END_IF
END_FUNCTION_BLOCK
ACTION CachePointers:
;
END_ACTION
ACTION CheckUpdateFlags:
xDataInUpdated := TRUE;
END_ACTION
ACTION DataReceived:
cmd := InDataTelegram_Module_1[0];
IF (cmd = M2C_NVI_UPDT_OCCD) OR (cmd = M2C_NV_VALUE_RSP) OR (cmd = M2C_NVI_UPDT_TOUT) THEN
	bNvRelativeIdx := (InDataTelegram_Module_1[1] - bNvStartIndex - bObjectIndex) / bLmoCount;
	CASE bNvRelativeIdx OF

	END_CASE
ELSIF (cmd = M2C_CP_VALUE_RSP) THEN
	wCpRelativeIdx := ((InDataTelegram_Module_1[1] + InDataTelegram_Module_1[2] * 256) - wCpStartIndex - bObjectIndex) / bLmoCount;
	CASE wCpRelativeIdx OF

	END_CASE
END_IF
END_ACTION
ACTION ResetNviUpdate:
;
END_ACTION
ACTION SendValueRequest:
;
END_ACTION
ACTION SetUpdateFlags:
;
END_ACTION

(* POU Plant/SCA_Proc, ST *)
PROGRAM SCA_Proc
VAR
	SCA01_1	:	FLT_TAP;
	SCA01_2	:	FLT_TAP;
	SCA01_3	:	FLT_TAP;

	upd		:	BOOL;
END_VAR
(***** SCA01 *****)
SCA01_1(IN:=SCA01_1_DI);
IF SCA01_1.EVL THEN LogEv(EL_Wrn,EO_SCA,1,1,'1'); upd:=TRUE; END_IF
IF SCA01_1.EVH THEN	LogEv(EL_Log,EO_SCA,1,2,'1'); upd:=TRUE; END_IF

SCA01_2(IN:=SCA01_2_DI);
IF SCA01_2.EVL THEN	LogEv(EL_Wrn,EO_SCA,1,1,'2'); upd:=TRUE; END_IF
IF SCA01_2.EVH THEN	LogEv(EL_Log,EO_SCA,1,2,'2'); upd:=TRUE; END_IF

SCA01_3(IN:=SCA01_3_DI);
IF SCA01_3.EVL THEN	LogEv(EL_Wrn,EO_SCA,1,1,'3'); upd:=TRUE; END_IF
IF SCA01_3.EVH THEN	LogEv(EL_Log,EO_SCA,1,2,'3'); upd:=TRUE; END_IF

IF upd THEN
	upd:=FALSE;
	Logger_Head();
	AddLogData();
	Logger_Send();
END_IF
END_PROGRAM
ACTION AddLogData:
Logger.s1:='&SCA01=';
Logger.s1:=CONCAT(Logger.s1,BYTE_TO_STRING(BOOL_TO_BYTE(SCA01_1.OUT))		); Logger.s1:=CONCAT(Logger.s1,';');
Logger.s1:=CONCAT(Logger.s1,BYTE_TO_STRING(BOOL_TO_BYTE(SCA01_2.OUT))		); Logger.s1:=CONCAT(Logger.s1,';');
Logger.s1:=CONCAT(Logger.s1,BYTE_TO_STRING(BOOL_TO_BYTE(SCA01_3.OUT))		);
ADDSTRING(ADR(Logger.TData), ADR(Logger.s1), Logger.TLen);
END_ACTION

(* POU TCP_Logger/LogEv, ST *)
FUNCTION LogEv : BOOL
VAR_INPUT
	Level	: en_Logger_ErrLev;
	Object  : en_SYS_Objects;
	Index	: WORD;
	Error	: WORD;
	Message : STRING;
END_VAR
VAR
	s1 : STRING(160);
	i  : INT;
END_VAR
(* Execute error level operations *)
CASE Level OF
	EL_Wrn: 		Sys.Warning:=TRUE;
	EL_Alarm: 		Sys.Alarm  :=TRUE;
	EL_AlarmStop: 	Sys.Alarm  :=TRUE; (* GO TO STOP STATE!! *)
END_CASE

(* Fill lastlog list *)
s1:=CONCAT(Sys.Time_LogString,';Lev=');
s1:=CONCAT(s1,INT_TO_STRING(Level));
s1:=CONCAT(s1,';Obj=');
s1:=CONCAT(s1,INT_TO_STRING(Object));
s1:=CONCAT(s1,';Idx=');
s1:=CONCAT(s1,WORD_TO_STRING(Index));
s1:=CONCAT(s1,';Err=');
s1:=CONCAT(s1,WORD_TO_STRING(Error));
Sys.LastLogs_Dat[Sys.LastLogs_Idx]:=s1;
Sys.LastLogs_Msg[Sys.LastLogs_Idx]:=Message;
Sys.LastLogs_Idx:=Sys.LastLogs_Idx+1;
IF Sys.LastLogs_Idx>5 THEN Sys.LastLogs_Idx:=0; END_IF

(*---------------------------------------------------------------*)
	Logger_Head();
(*---------------------------------------------------------------*)

(* Insert ERR *)
s1:=CONCAT('&ERR=',INT_TO_STRING(Level));
s1:=CONCAT(s1,';');
s1:=CONCAT(s1,INT_TO_STRING(Object));
s1:=CONCAT(s1,';');
s1:=CONCAT(s1,WORD_TO_STRING(Index));
s1:=CONCAT(s1,';');
s1:=CONCAT(s1,WORD_TO_STRING(Error));
s1:=CONCAT(s1,';');
ADDSTRING(ADR(Logger.TData), ADR(s1), Logger.TLen);
s1:=Message;
STR_NOSPACES(ADR(s1));
ADDSTRING(ADR(Logger.TData), ADR(s1), Logger.TLen);

(*---------------------------------------------------------------*)
	Logger_Send();
(*---------------------------------------------------------------*)
END_FUNCTION

(* POU TCP_Logger/Logger_Head, ST *)
FUNCTION Logger_Head : BOOL
VAR
	s1 : STRING(160);
	i  : BYTE;
END_VAR
Logger.TLen:=0;
(* Set GET header *)
ADDSTRING(ADR(Logger.TData), ADR(Logger_GETSTART), Logger.TLen);

(* Insert Header *)
s1:=INSERT('ID=&V=1&D=',DWORD_TO_STRING(Plant_SN),3);
s1:=CONCAT(s1,Sys.Time_LogString);
s1:=CONCAT(s1,'&S=');
IF Sys.Alarm THEN i:=2; ELSIF Sys.Warning THEN i:=1; ELSE i:=0; END_IF
s1:=CONCAT(s1,BYTE_TO_STRING(i));
ADDSTRING(ADR(Logger.TData), ADR(s1), Logger.TLen);
END_FUNCTION

(* POU Utils Functions/ADDSTRING, ST *)
FUNCTION ADDSTRING : BOOL (* Append string to a byte buffer *)
VAR_INPUT
	pTxData: POINTER TO BYTE;
	pString: POINTER TO BYTE;
END_VAR
VAR_IN_OUT
	TxLen: DINT;
END_VAR
VAR
END_VAR
pTxData:=pTxData+TxLen;
WHILE pString^<>0 DO
	pTxData^:=pString^;
	pString:=pString+1;
	pTxData:=pTxData+1;
	TxLen:=TxLen+1;
END_WHILE
END_FUNCTION

(* POU Utils Functions/STR_NOSPACES, ST *)
FUNCTION STR_NOSPACES : BOOL (* Replace spaces and bad chars with allowed ones, used as HTTP-GET validator *)
VAR_INPUT
	pString: POINTER TO BYTE;
END_VAR
VAR
END_VAR
WHILE pString^<>0 DO
	IF pString^=16#20 (* space *) THEN pString^:=16#5F; (*'_'*) END_IF
	pString:=pString+1;
END_WHILE
END_FUNCTION

(* POU TCP_Logger/Logger_Send, ST *)
FUNCTION Logger_Send : BOOL
VAR
	hFile: 	DWORD;
	pos:	DWORD;
END_VAR
(* Finalize string *)
ADDSTRING(ADR(Logger.TData), ADR(Logger_GETEND), Logger.TLen);

(* Read log position *)
pos:=SysFileGetSize(Logger_DataFile);
(* Check log size, bckup and erase if no pending messages *)
IF pos>5000000(*5M*) THEN
	hFile:=SysFileOpen(Logger_IndexFile,'r');
	IF hFile=0 THEN
		SysFileDelete(Logger_DataFileOld);
		SysFileRename(Logger_DataFile,Logger_DataFileOld);
		pos:=0;
	ELSE
		SysFileClose(hFile);
	END_IF
END_IF
(* Write message on log file *)
hFile:=SysFileOpen(Logger_DataFile,'a');
IF hFile<>0 THEN
	SysFileWrite(hFile, ADR(Logger.TData), Logger.TLen);
	SysFileClose(hFile);
ELSE
	Sys.Warning:=TRUE;
END_IF


(* Check logger status *)
IF Logger.SendReq=FALSE THEN
	(* Set log position for recovery *)
	Logger.SendIdx:=pos;
	(* Copy message data *)
	MEMCPY(ADR(Logger.TData),ADR(Logger.SendData),DINT_TO_WORD(Logger.TLen));
	Logger.SendLen:=Logger.TLen;
	(* Trigger request *)
	Logger.SendReq:=TRUE;
ELSE
	(* Add message position+size in recovery indexes *)
	hFile:=SysFileOpen(Logger_IndexFile,'a');
	SysFileWrite(hFile, ADR(pos), SIZEOF(pos));
	SysFileWrite(hFile, ADR(Logger.TLen), SIZEOF(Logger.TLen));
	SysFileClose(hFile);
END_IF
END_FUNCTION

(* POU Utils Functions/MEMCPY, ST *)
FUNCTION MEMCPY:BOOL
VAR_INPUT
	pSourceAddress:POINTER TO ARRAY[1..2] OF BYTE;
	pDestinationAddress:POINTER TO ARRAY[1..2] OF BYTE;
	BytesToCopy:WORD;
END_VAR
VAR
END_VAR
WHILE (BytesToCopy > 0) DO
	pDestinationAddress^[1]:=pSourceAddress^[1]; (* copy bytes from source to destination *)
	pDestinationAddress:=ADR(pDestinationAddress^[2]); (* increment destination *)
	pSourceAddress:=ADR(pSourceAddress^[2]);(* increment source *)
	BytesToCopy:=BytesToCopy -1; (* decrement number of bytes to copy *)
END_WHILE
END_FUNCTION

(* POU Plant/SYS_Proc, ST *)
PROGRAM SYS_Proc
VAR
(*	fALARM_PB		:FLT_TAP;
	fALARM_TB		:FLT_TAP;
	fALARM_PM		:FLT_TAP; *)

(*	fGZB_ST			:FLT_TAP; (* GATEWAY ZIGBEE *)*)
(*	fVPN_OUT1		:FLT_TAP; (* VPN - CONNECT *)*)
	fVPN_OUT2		:FLT_TAP; (* VPN - STATUS *)
(*	fKEY_CT_ST		:FLT_TAP; (* DOOR01 - Porta primaria *)*)
(*	fKEY_SCT_ST		:FLT_TAP; (* DOOR02 - Porta secondaria *)*)
	fKEY_QE_ST		:FLT_TAP; (* DOOR03 - Quadro Elettrico *)
	fKEY_ManualMode :FLT_TAP; (* Selettore Luci in manuale *)

END_VAR
(*************** ISPESL *****************)
(*
fALARM_PB(IN:=ALARM_PB);
IF fALARM_PB.EVH THEN
	LogEv(EL_AlarmStop,EO_PBV,1,1,'Over_Pressure_Alarm');
END_IF

fALARM_TB(IN:=ALARM_TB);
IF fALARM_TB.EVH THEN
	LogEv(EL_AlarmStop,EO_TBV,1,1,'Over_Temperature_Alarm');
END_IF

fALARM_PM(IN:=ALARM_PM);
IF fALARM_PM.EVH THEN
	LogEv(EL_AlarmStop,EO_PMV,1,1,'Under_Pressure_Alarm');
END_IF
*)
(****************************************)

(*### VPN Connection Check ###*)(*
fVPN_OUT1(IN:=VPN_OUT1);
IF fVPN_OUT1.EVH THEN
	LogEv(EL_Log,EO_VPN,1,1,'CONNECT_ON');
END_IF
IF fVPN_OUT1.EVL THEN
	LogEv(EL_Log,EO_VPN,1,2,'CONNECT_OFF');
END_IF*)

(*### VPN Status Check ###*)
fVPN_OUT2(IN:=VPN_OUT2);
IF fVPN_OUT2.EVH THEN
	LogEv(EL_Log,EO_VPN,1,3,'STATUS_UP');
END_IF
IF fVPN_OUT2.EVL THEN
	LogEv(EL_Wrn,EO_VPN,1,4,'STATUS_DOWN');
END_IF

(*### DOOR01 Status Check ###*)(*
fKEY_CT_ST(IN:=KEY_CT_ST);
IF fKEY_CT_ST.EVH THEN
	LogEv(EL_Log,EO_DOOR,1,2,'Centrale_termica_Close');
END_IF
IF fKEY_CT_ST.EVL THEN
	LogEv(EL_Wrn,EO_DOOR,1,1,'Centrale_termica_Open');
END_IF*)

(*### DOOR02 Status Check ###*)(*
fKEY_SCT_ST(IN:=KEY_SCT_ST);
IF fKEY_SCT_ST.EVH THEN
	LogEv(EL_Log,EO_DOOR,2,2,'Sottocentrale_termica_Close');
END_IF
IF fKEY_SCT_ST.EVL THEN
	LogEv(EL_Wrn,EO_DOOR,2,1,'Sottocentrale_termica_Open');
END_IF*)

(*### DOOR03 Status Check ###*)
fKEY_QE_ST(IN:=KEY_QE_ST);
IF fKEY_QE_ST.EVH THEN
	LogEv(EL_Log,EO_DOOR,3,2,'Quadro_Close');
END_IF
IF fKEY_QE_ST.EVL THEN
	LogEv(EL_Wrn,EO_DOOR,3,1,'Quadro_Open');
END_IF

(*### Selettore luci in manuale ###*)
fKEY_ManualMode(IN:=SCA01_1_DI);
IF fKEY_ManualMode.EVH THEN
	LogEv(EL_Alarm,EO_LUX,0,10,'Impianto_in Manuale');
END_IF
IF fKEY_ManualMode.EVL THEN
	LogEv(EL_Log,EO_LUX,0,11,'Impianto_In_Automatico');
END_IF
END_PROGRAM

(* POU Utils Functions/AVERAGE_T, ST *)
FUNCTION_BLOCK AVERAGE_T
VAR_INPUT
	IN: 	INT;
END_VAR
VAR_OUTPUT
	HI:		INT;
	AVG:	INT;
	LOW:	INT;
	ERR:	BOOL;
END_VAR
VAR
	sum:	DINT;
	cnt:	WORD;
END_VAR
IF cnt>=65000 THEN
	ERR:=TRUE;
	Read();
	sum := sum - AVG;
	cnt := cnt + 1;
END_IF

sum := sum + IN;
cnt := cnt + 1;

IF IN<LOW THEN  LOW:=IN; END_IF
IF IN>HI  THEN HI :=IN; END_IF
END_FUNCTION_BLOCK
ACTION Read:
AVG := DINT_TO_INT(sum/cnt);
END_ACTION
ACTION Reset:
HI:=IN;
AVG:=IN;
LOW:=IN;
ERR:=FALSE;

sum:=IN;
cnt:=1;
END_ACTION

(* POU Utils Functions/BUILD_16TO32, ST *)
FUNCTION BUILD_16TO32 : DWORD
VAR_INPUT
		pSource	:	POINTER TO WORD;
END_VAR
VAR
		Data	:	DWORD;
END_VAR
Data := WORD_TO_DWORD(pSource^);
pSource := pSource + 1;
Data := Data + WORD_TO_DWORD(pSource^) * 65536;

BUILD_16TO32 := Data;
END_FUNCTION

(* POU Utils Functions/COPY_32SWAP16, ST *)
FUNCTION COPY_32SWAP16:BOOL
VAR_INPUT
	pSourceAddress		:POINTER TO ARRAY[1..2] OF WORD;
	pDestinationAddress	:POINTER TO ARRAY[1..2] OF WORD;
END_VAR
VAR
END_VAR
pDestinationAddress^[1]:=pSourceAddress^[2];
pDestinationAddress^[2]:=pSourceAddress^[1];
END_FUNCTION

(* POU Utils Functions/FLT_KEY, ST *)
FUNCTION_BLOCK FLT_KEY
VAR_INPUT
	IN		: BOOL;
	TTAP	: TIME:=T#5s;
	INITEV	: BOOL:=TRUE;
END_VAR
VAR_OUTPUT
	OUT		: BOOL;
	EVH		: BOOL;
	EVL		: BOOL;
END_VAR
VAR
	init	: BOOL:=FALSE;
	timer	: TON;
	timerIn	: TON;				(* Inhibition timer *)
	fInhibit: BOOL:=FALSE;
END_VAR
EVH:=FALSE;
EVL:=FALSE;

IF NOT init THEN
	init := TRUE;
	IF INITEV THEN
		OUT  := NOT IN;
	ELSE
		OUT  := IN;
	END_IF
END_IF

timerIn(IN:=fInhibit,PT:=T#500ms);

IF timerIn.Q THEN fInhibit := FALSE; END_IF

IF NOT fInhibit THEN

	IF OUT<>IN THEN
		timer(IN:=TRUE,PT:=TTAP);
		IF timer.Q THEN
			OUT:=IN;
			timer(IN:=FALSE);
			fInhibit := TRUE;
			IF OUT THEN EVH:=TRUE; ELSE EVL:=TRUE; END_IF
		END_IF
	ELSE
		timer(IN:=FALSE);
	END_IF
END_IF
END_FUNCTION_BLOCK

(* POU Utils Functions/FLT_TIME, ST *)
FUNCTION_BLOCK FLT_TIME
VAR_INPUT
	IN		: BOOL;
	TTAP	: TIME:=T#5s;
	INITEV	: BOOL:=TRUE;
END_VAR
VAR_OUTPUT
	OUT		: BOOL;
	EVH		: BOOL;
	EVL		: BOOL;
END_VAR
VAR
	init	: BOOL:=FALSE;
	timer	: TON;
END_VAR
EVH:=FALSE;
EVL:=FALSE;

IF NOT init THEN
	init := TRUE;
	IF INITEV THEN
		OUT  := NOT IN;
	ELSE
		OUT  := IN;
	END_IF
END_IF

IF OUT<>IN THEN
	timer(IN:=TRUE,PT:=TTAP);
	IF timer.Q THEN
		OUT:=IN;
		timer(IN:=FALSE);
		IF OUT THEN EVH:=TRUE; ELSE EVL:=TRUE; END_IF
	END_IF
ELSE
	timer(IN:=FALSE);
END_IF
END_FUNCTION_BLOCK

(* POU LON/Module_1/Internal/FuDoCpUpdate_Module_1, ST *)
FUNCTION FuDoCpUpdate_Module_1 : BOOL
(******************************************)
(* Automatic generated code, do not edit! *)
(******************************************)
VAR_INPUT
	ptCp : POINTER TO BYTE;
	ptCpLast : POINTER TO BYTE;
	wCpIndex : WORD;
	uiCpLength : UINT;
	uiCpVariableLength : UINT;
END_VAR
OutDataTelegram_Module_1[0] := C2M_CP_VALUE;
OutDataTelegram_Module_1[1] := WORD_TO_BYTE(wCpIndex AND 16#FF);
OutDataTelegram_Module_1[2] := WORD_TO_BYTE((wCpIndex / 256) AND 16#FF);

mbxModule_1.bTxPrio := 1;
mbxModule_1.bTxProtID := 0;
mbxModule_1.pbTxData := ADR(OutDataTelegram_Module_1);
mbxModule_1.unTxLen := 3 + uiCpLength;
mbxModule_1.MBX_SEND();

IF (mbxModule_1.nError <> MBX_OK) THEN
	FuDoCpUpdate_Module_1 := FALSE;
	RETURN;
END_IF

FuMemCopy(ptCp, ptCpLast, uiCpVariableLength);

FuDoCpUpdate_Module_1 := TRUE;
END_FUNCTION

(* POU LON/Shared/Internal/FuRawToSnvtFilePos, ST *)
FUNCTION FuRawToSnvtFilePos : BOOL
(******************************************)
(* Automatic generated code, do not edit! *)
(******************************************)
VAR_INPUT
	RawDataIn : POINTER TO ARRAY[0..5] OF BYTE;
	DataOut : POINTER TO typSnvtFilePos;
END_VAR
VAR
END_VAR
DataOut^.diRwPtr := RawDataIn^[0] * 16777216 + RawDataIn^[1] * 65536 + RawDataIn^[2] * 256 + RawDataIn^[3];

DataOut^.wRwLength := RawDataIn^[4] * 256 + RawDataIn^[5];

FuRawToSnvtFilePos := TRUE;
END_FUNCTION

(* POU LON/Shared/Internal/FuRawToSnvtFileReq, ST *)
FUNCTION FuRawToSnvtFileReq : BOOL
(******************************************)
(* Automatic generated code, do not edit! *)
(******************************************)
VAR_INPUT
	RawDataIn : POINTER TO ARRAY[0..11] OF BYTE;
	DataOut : POINTER TO typSnvtFileReq;
END_VAR
VAR
END_VAR
DataOut^.bRequest := RawDataIn^[0];

DataOut^.wIndex := RawDataIn^[1] * 256 + RawDataIn^[2];

DataOut^.wReceiveTimeout := RawDataIn^[3] * 256 + RawDataIn^[4];

DataOut^.abDestAddress[0] := RawDataIn^[5];
DataOut^.abDestAddress[1] := RawDataIn^[6];
DataOut^.abDestAddress[2] := RawDataIn^[7];
DataOut^.abDestAddress[3] := RawDataIn^[8];
DataOut^.abDestAddress[4] := RawDataIn^[9];

DataOut^.bAuthOn := RawDataIn^[10];

DataOut^.bPrioOn := RawDataIn^[11];

FuRawToSnvtFileReq := TRUE;
END_FUNCTION

(* POU LON/Shared/Internal/FuRawToSnvtFileStatus, ST *)
FUNCTION FuRawToSnvtFileStatus : BOOL
(******************************************)
(* Automatic generated code, do not edit! *)
(******************************************)
VAR_INPUT
	RawDataIn : POINTER TO ARRAY[0..26] OF BYTE;
	DataOut : POINTER TO typSnvtFileStatus;
END_VAR
VAR
END_VAR
DataOut^.bStatus := RawDataIn^[0];

DataOut^.wNumberOfFiles := RawDataIn^[1] * 256 + RawDataIn^[2];

DataOut^.wSelectedFile := RawDataIn^[3] * 256 + RawDataIn^[4];

DataOut^.abAdr[0] := RawDataIn^[5];
DataOut^.abAdr[1] := RawDataIn^[6];
DataOut^.abAdr[2] := RawDataIn^[7];
DataOut^.abAdr[3] := RawDataIn^[8];
DataOut^.abAdr[4] := RawDataIn^[9];
DataOut^.abAdr[5] := RawDataIn^[10];
DataOut^.abAdr[6] := RawDataIn^[11];
DataOut^.abAdr[7] := RawDataIn^[12];
DataOut^.abAdr[8] := RawDataIn^[13];
DataOut^.abAdr[9] := RawDataIn^[14];
DataOut^.abAdr[10] := RawDataIn^[15];
DataOut^.abAdr[11] := RawDataIn^[16];
DataOut^.abAdr[12] := RawDataIn^[17];
DataOut^.abAdr[13] := RawDataIn^[18];
DataOut^.abAdr[14] := RawDataIn^[19];
DataOut^.abAdr[15] := RawDataIn^[20];
DataOut^.abAdr[16] := RawDataIn^[21];
DataOut^.abAdr[17] := RawDataIn^[22];
DataOut^.abAdr[18] := RawDataIn^[23];
DataOut^.abAdr[19] := RawDataIn^[24];
DataOut^.abAdr[20] := RawDataIn^[25];
DataOut^.abAdr[21] := RawDataIn^[26];

FuRawToSnvtFileStatus := TRUE;
END_FUNCTION

(* POU LON/Shared/Internal/FuRawToSnvtObjRequest, ST *)
FUNCTION FuRawToSnvtObjRequest : BOOL
(******************************************)
(* Automatic generated code, do not edit! *)
(******************************************)
VAR_INPUT
	RawDataIn : POINTER TO ARRAY[0..2] OF BYTE;
	DataOut : POINTER TO typSnvtObjRequest;
END_VAR
VAR
END_VAR
DataOut^.wObjectId := RawDataIn^[0] * 256 + RawDataIn^[1];

DataOut^.bObjectRequest := RawDataIn^[2];

FuRawToSnvtObjRequest := TRUE;
END_FUNCTION

(* POU LON/Shared/Internal/FuRawToSnvtObjStatus, ST *)
FUNCTION FuRawToSnvtObjStatus : BOOL
(******************************************)
(* Automatic generated code, do not edit! *)
(******************************************)
VAR_INPUT
	RawDataIn : POINTER TO ARRAY[0..5] OF BYTE;
	DataOut : POINTER TO typSnvtObjStatus;
END_VAR
VAR
END_VAR
DataOut^.wObjectId := RawDataIn^[0] * 256 + RawDataIn^[1];

DataOut^.bBitfieldByteOffset2 := RawDataIn^[2];

DataOut^.bBitfieldByteOffset3 := RawDataIn^[3];

DataOut^.bBitfieldByteOffset4 := RawDataIn^[4];

DataOut^.bBitfieldByteOffset5 := RawDataIn^[5];

FuRawToSnvtObjStatus := TRUE;
END_FUNCTION

(* POU LON/Module_1/Internal/FuSendCpValueReq_Module_1, ST *)
FUNCTION FuSendCpValueReq_Module_1 : BOOL
(******************************************)
(* Automatic generated code, do not edit! *)
(******************************************)
VAR_INPUT
	ptCp : POINTER TO BYTE;
	ptInternalUseOnly : POINTER TO BYTE;
	wCpIndex : WORD;
END_VAR
IF (ptCp <> 0) THEN
	IF ptInternalUseOnly^.0 = TRUE THEN
		OutDataTelegram_Module_1[0] := C2M_CP_VALUE_QRY;
		OutDataTelegram_Module_1[1] := WORD_TO_BYTE(wCpIndex AND 16#FF);
		OutDataTelegram_Module_1[2] := WORD_TO_BYTE((wCpIndex / 256) AND 16#FF);

		mbxModule_1.bTxPrio := 1;
		mbxModule_1.bTxProtID := 0;
		mbxModule_1.pbTxData := ADR(OutDataTelegram_Module_1);
		mbxModule_1.unTxLen := 3;
		mbxModule_1.MBX_SEND();

		IF (mbxModule_1.nError <> MBX_OK) THEN
			FuSendCpValueReq_Module_1 := FALSE;
			RETURN;
		END_IF
		ptInternalUseOnly^.0 := FALSE;
	END_IF
END_IF

FuSendCpValueReq_Module_1 := TRUE;
END_FUNCTION

(* POU LON/Shared/Internal/FuSnvtFilePosToRaw, ST *)
FUNCTION FuSnvtFilePosToRaw : BOOL
(******************************************)
(* Automatic generated code, do not edit! *)
(******************************************)
VAR_INPUT
	NvDataIn :  POINTER TO typSnvtFilePos;
	DataOut : POINTER TO ARRAY[0..5] OF BYTE;
END_VAR
VAR
END_VAR
DataOut^[0] := DINT_TO_BYTE(SHR(NvDataIn^.diRwPtr, 24));
DataOut^[1] := DINT_TO_BYTE(SHR(NvDataIn^.diRwPtr, 16));
DataOut^[2] := DINT_TO_BYTE(SHR(NvDataIn^.diRwPtr, 8));
DataOut^[3] := DINT_TO_BYTE(NvDataIn^.diRwPtr);

DataOut^[4] := WORD_TO_BYTE(SHR(NvDataIn^.wRwLength, 8));
DataOut^[5] := WORD_TO_BYTE(NvDataIn^.wRwLength);

FuSnvtFilePosToRaw := TRUE;
END_FUNCTION

(* POU LON/Shared/Internal/FuSnvtFileReqToRaw, ST *)
FUNCTION FuSnvtFileReqToRaw : BOOL
(******************************************)
(* Automatic generated code, do not edit! *)
(******************************************)
VAR_INPUT
	NvDataIn :  POINTER TO typSnvtFileReq;
	DataOut : POINTER TO ARRAY[0..11] OF BYTE;
END_VAR
VAR
END_VAR
DataOut^[0] := NvDataIn^.bRequest;

DataOut^[1] := WORD_TO_BYTE(SHR(NvDataIn^.wIndex, 8));
DataOut^[2] := WORD_TO_BYTE(NvDataIn^.wIndex);

DataOut^[3] := WORD_TO_BYTE(SHR(NvDataIn^.wReceiveTimeout, 8));
DataOut^[4] := WORD_TO_BYTE(NvDataIn^.wReceiveTimeout);

DataOut^[5] := NvDataIn^.abDestAddress[0];
DataOut^[6] := NvDataIn^.abDestAddress[1];
DataOut^[7] := NvDataIn^.abDestAddress[2];
DataOut^[8] := NvDataIn^.abDestAddress[3];
DataOut^[9] := NvDataIn^.abDestAddress[4];

DataOut^[10] := NvDataIn^.bAuthOn;

DataOut^[11] := NvDataIn^.bPrioOn;

FuSnvtFileReqToRaw := TRUE;
END_FUNCTION

(* POU LON/Shared/Internal/FuSnvtObjRequestToRaw, ST *)
FUNCTION FuSnvtObjRequestToRaw : BOOL
(******************************************)
(* Automatic generated code, do not edit! *)
(******************************************)
VAR_INPUT
	NvDataIn :  POINTER TO typSnvtObjRequest;
	DataOut : POINTER TO ARRAY[0..2] OF BYTE;
END_VAR
VAR
END_VAR
DataOut^[0] := WORD_TO_BYTE(SHR(NvDataIn^.wObjectId, 8));
DataOut^[1] := WORD_TO_BYTE(NvDataIn^.wObjectId);

DataOut^[2] := NvDataIn^.bObjectRequest;

FuSnvtObjRequestToRaw := TRUE;
END_FUNCTION

(* POU TCP_Logger/LogTrig, ST *)
FUNCTION LogTrig : BOOL
VAR
	s1 : STRING(160);
	i  : BYTE;
END_VAR
(*---------------------------------------------------------------*)
	Logger_Head();
(*---------------------------------------------------------------*)

(* Insert contabilizers  *)
ANZ01.AddLogData( ModBus:=MODB01 );
ANZ02.AddLogData( ModBus:=MODB01 );
HVAC01.AddLogData(ModBus:=MODB02);
HVAC02.AddLogData(ModBus:=MODB02);

COOV01.AddLogData();

LUX01.AddLogData(WORKINGTIME:=LuxWT[1], POWERONCYCLES:=LuxPOC[1]);
LUX02.AddLogData(WORKINGTIME:=LuxWT[2], POWERONCYCLES:=LuxPOC[2]);
LUX03.AddLogData(WORKINGTIME:=LuxWT[3], POWERONCYCLES:=LuxPOC[3]);
LUX04.AddLogData(WORKINGTIME:=LuxWT[4], POWERONCYCLES:=LuxPOC[4]);
LUX05.AddLogData(WORKINGTIME:=LuxWT[5], POWERONCYCLES:=LuxPOC[5]);
LUX06.AddLogData(WORKINGTIME:=LuxWT[6], POWERONCYCLES:=LuxPOC[6]);

ZTHL01.AddLogData(ModBus:=MODB03);
ZTHL02.AddLogData(ModBus:=MODB03);
ZTHL03.AddLogData(ModBus:=MODB03);
ZTHL04.AddLogData(ModBus:=MODB03);


(*---------------------------------------------------------------*)
	Logger_Send();
(*---------------------------------------------------------------*)
END_FUNCTION

(* POU Utils Functions/MEAN_VALUE, ST *)
FUNCTION MEAN_VALUE : WORD
VAR_INPUT
		pArray	:	POINTER TO ARRAY [1..2] OF WORD;
		Length	:	WORD;
END_VAR
VAR
		counter	:	WORD;
		Sum		:	DWORD;
		(*Maximum	:	WORD;
		Minimum	:	WORD;*)
END_VAR
Sum := 0;
(*Maximum := 0;
Minimum := 0;*)

FOR counter:=1 TO Length BY 1 DO
	Sum := Sum + WORD_TO_DWORD(pArray^[counter]);

	(*IF pArray^[counter] > Maximum THEN Maximum := pArray^[counter]; END_IF
	IF pArray^[counter] < Minimum THEN Minimum := pArray^[counter]; END_IF*)

END_FOR

(*Sum := Sum - WORD_TO_DWORD(Maximum) - WORD_TO_DWORD(Minimum);
MEAN_VALUE := DWORD_TO_WORD(Sum/(Length-2));*)

MEAN_VALUE := DWORD_TO_WORD(Sum/Length);
END_FUNCTION

(* POU Utils Functions/MEMCLR, ST *)
FUNCTION MEMCLR:BOOL
VAR_INPUT
	pDestinationAddress:POINTER TO ARRAY[1..2] OF BYTE;
	BytesToClear:WORD;
END_VAR
VAR
END_VAR
WHILE (BytesToClear > 0) DO
	pDestinationAddress^[1]:=0;
	pDestinationAddress:=ADR(pDestinationAddress^[2]); (* increment destination *)
	BytesToClear:=BytesToClear -1; (* decrement number of bytes to copy *)
END_WHILE
END_FUNCTION

(* POU LON/Module_1/ApplicationMessage/Module_1_ApplicationMsgSend, ST *)
FUNCTION_BLOCK Module_1_ApplicationMsgSend
(******************************************)
(* Automatic generated code, do not edit! *)
(******************************************)
VAR_INPUT
	xSend 		  : BOOL;
	abAddress     : ARRAY[0..10] OF BYTE;
	typServiceSend  : ServiceType;
	xPriority : BOOL;
	xAuthentification : BOOL;
	bMsgCodeSend  : BYTE;
	abMsgDataSend : ARRAY[0..47] OF BYTE;
	bLengthSend	  : BYTE;
END_VAR
VAR_OUTPUT
	bSendStatus   : BYTE;
END_VAR
VAR
	bAddressLength : BYTE;
	RtrigSend : R_TRIG;
END_VAR
RtrigSend(CLK:=xSend);
IF RtrigSend.Q AND (xInitRunning_Module_1 = FALSE) AND (mbxModule_1.bStatus.0) THEN
	OutDataTelegram_Module_1[0] := C2M_LON_MSG_SEND;
	OutDataTelegram_Module_1[1] := INT_TO_BYTE(typServiceSend);
	OutDataTelegram_Module_1[1].6 := xAuthentification;
	OutDataTelegram_Module_1[1].7 := xPriority;
	IF (abAddress[0] = 2) THEN
		bAddressLength := 11;
	ELSE
		bAddressLength := 5;
	END_IF
	FuMemCopy(ADR(abAddress), ADR(OutDataTelegram_Module_1[2]), bAddressLength);
	OutDataTelegram_Module_1[2+bAddressLength] := bMsgCodeSend;
	IF bLengthSend > 48 THEN bLengthSend := 48; END_IF;
	FuMemCopy(ADR(abMsgDataSend), ADR(OutDataTelegram_Module_1[2+bAddressLength+1]), bLengthSend);

	mbxModule_1.bTxPrio := BOOL_TO_BYTE(xPriority);
	mbxModule_1.bTxProtID := 0;
	mbxModule_1.pbTxData := ADR(OutDataTelegram_Module_1);
	mbxModule_1.unTxLen := 3 + bAddressLength + bLengthSend;
	mbxModule_1.MBX_SEND();

	IF (mbxModule_1.nError <> MBX_OK) THEN
		bSendStatus := 255;
	ELSE
		bSendStatus := 0;
	END_IF
END_IF
END_FUNCTION_BLOCK

(* POU LON/Module_1/ApplicationMessage/Module_1_ApplicationMsgSendRsp, ST *)
FUNCTION_BLOCK Module_1_ApplicationMsgSendRsp
(******************************************)
(* Automatic generated code, do not edit! *)
(******************************************)
VAR_INPUT
	xSend 	  : BOOL;
	bCorrelator : BYTE;
	bMsgCode  : BYTE;
	abMsgData : ARRAY[0..47] OF BYTE;
	bLength	  : BYTE;
END_VAR
VAR_OUTPUT
	bSendStatus : BYTE;
END_VAR
VAR
	RtrigSend : R_TRIG;
END_VAR
RtrigSend(CLK:=xSend);
IF RtrigSend.Q AND (xInitRunning_Module_1 = FALSE) AND (mbxModule_1.bStatus.0) THEN
	OutDataTelegram_Module_1[0] := C2M_LON_MSG_RSP_SEND;
	OutDataTelegram_Module_1[1] := bCorrelator;
	OutDataTelegram_Module_1[2] := bMsgCode;
	IF bLength > 48 THEN bLength := 48; END_IF;
	FuMemCopy(ADR(abMsgData), ADR(OutDataTelegram_Module_1[3]), bLength);

	mbxModule_1.bTxPrio := BOOL_TO_BYTE(bCorrelator.7);
	mbxModule_1.bTxProtID := 0;
	mbxModule_1.pbTxData := ADR(OutDataTelegram_Module_1);
	mbxModule_1.unTxLen := 3 + bLength;
	mbxModule_1.MBX_SEND();

	IF (mbxModule_1.nError <> MBX_OK) THEN
		bSendStatus := 255;
	ELSE
		bSendStatus := 0;
	END_IF
END_IF
END_FUNCTION_BLOCK

(* POU Plant_Objects/obj_COO, ST *)
FUNCTION_BLOCK obj_COO
(* === CO2 SENSOR ===
   v1.0[29/09/15] - Versioning
*)
VAR_INPUT
	ID			:	BYTE;

	In1			:	WORD;
	In2			:	WORD;
	In3			:	WORD;
	In4			:	WORD;
	In5			:	WORD;

	ProbesNr	:	BYTE;
END_VAR
VAR_OUTPUT
	Out1		:	WORD;
	Out2		:	WORD;
	Out3		:	WORD;
	Out4		:	WORD;
	Out5		:	WORD;

	Status_Log	:	WORD;
END_VAR
VAR
	i			:	BYTE;
END_VAR
(* Copy active input(s) to output(s)	*)
CASE ProbesNr OF

	1:
		Out1 := In1;

	2:
		Out1 := In1;
		Out2 := In2;

	3:
		Out1 := In1;
		Out2 := In2;
		Out3 := In3;

	4:
		Out1 := In1;
		Out2 := In2;
		Out3 := In3;
		Out4 := In4;

	5:
		Out1 := In1;
		Out2 := In2;
		Out3 := In3;
		Out4 := In4;
		Out5 := In5;

END_CASE

Status_Log := 0;
END_FUNCTION_BLOCK
ACTION AddLogData:
Logger.s1:='&COOV=';

CASE ProbesNr OF

	1:
		Logger.s1:=CONCAT(Logger.s1,WORD_TO_STRING(In1));
		Logger.s1:=CONCAT(Logger.s1,';');

	2:
		Logger.s1:=CONCAT(Logger.s1,WORD_TO_STRING(In1));
		Logger.s1:=CONCAT(Logger.s1,';');
		Logger.s1:=CONCAT(Logger.s1,WORD_TO_STRING(In2));
		Logger.s1:=CONCAT(Logger.s1,';');

	3:
		Logger.s1:=CONCAT(Logger.s1,WORD_TO_STRING(In1));
		Logger.s1:=CONCAT(Logger.s1,';');
		Logger.s1:=CONCAT(Logger.s1,WORD_TO_STRING(In2));
		Logger.s1:=CONCAT(Logger.s1,';');
		Logger.s1:=CONCAT(Logger.s1,WORD_TO_STRING(In3));
		Logger.s1:=CONCAT(Logger.s1,';');

	4:
		Logger.s1:=CONCAT(Logger.s1,WORD_TO_STRING(In1));
		Logger.s1:=CONCAT(Logger.s1,';');
		Logger.s1:=CONCAT(Logger.s1,WORD_TO_STRING(In2));
		Logger.s1:=CONCAT(Logger.s1,';');
		Logger.s1:=CONCAT(Logger.s1,WORD_TO_STRING(In3));
		Logger.s1:=CONCAT(Logger.s1,';');
		Logger.s1:=CONCAT(Logger.s1,WORD_TO_STRING(In4));
		Logger.s1:=CONCAT(Logger.s1,';');

	5:
		Logger.s1:=CONCAT(Logger.s1,WORD_TO_STRING(In1));
		Logger.s1:=CONCAT(Logger.s1,';');
		Logger.s1:=CONCAT(Logger.s1,WORD_TO_STRING(In2));
		Logger.s1:=CONCAT(Logger.s1,';');
		Logger.s1:=CONCAT(Logger.s1,WORD_TO_STRING(In3));
		Logger.s1:=CONCAT(Logger.s1,';');
		Logger.s1:=CONCAT(Logger.s1,WORD_TO_STRING(In4));
		Logger.s1:=CONCAT(Logger.s1,';');
		Logger.s1:=CONCAT(Logger.s1,WORD_TO_STRING(In5));
		Logger.s1:=CONCAT(Logger.s1,';');

END_CASE


Logger.s1:=CONCAT(Logger.s1,WORD_TO_STRING(Status_Log));
ADDSTRING(ADR(Logger.TData), ADR(Logger.s1), Logger.TLen);
END_ACTION

(* POU Plant_Objects/obj_CRON, ST *)
FUNCTION_BLOCK obj_CRON
(* === CRONOGRAFO STANDARD ===
   v1.0[16/04/15] - Versioning
   v1.1[19/05/15] - Removed DB creation from previous year
*)
VAR_INPUT
	(* Settings *)
	ID			: BYTE;		(* Index of instanced object *)

	InitOK		: BOOL;
	Alarm		: BOOL;
	Warning		: BOOL;

	Profile		: typ_Cron_Profile; 				(* Profilo attivo *)
	ProfileNr	: BYTE;								(* Indice profilo attivo *)
	CalendarIdx : WORD;								(* Indice calendario attivo *)
	Jolly		: ARRAY[0..9] OF typ_Cron_Jolly;	(* Jolly attivi *)

END_VAR
VAR_IN_OUT
END_VAR
VAR_OUTPUT
	SetPoint		: INT;
	(* Status *)
	Status_Log		: BYTE;
	Status_Vis 		: DWORD;
END_VAR
VAR
	Buf: 	ARRAY[0..512] OF BYTE; (* AVOID THIS!! *)
	hFile: 	DWORD;
	sFile: 	STRING;
	sFile2: STRING;

	i:		WORD;
	t1:		DWORD;
	t2:		BOOL;

END_VAR
(* Check initialization *)
IF NOT InitOK THEN Init(); END_IF

(* Chrono *)
IF CalendarIdx<>Sys.Time_CT_Day THEN DB_Load(); END_IF
SetPoint:=Profile.Setpoint[Sys.Time_CT_Quarter];

(* Check jolly *)
FOR i := 0 TO 9 DO
	IF ( DT_TO_DWORD(Jolly[i].Start)>0  AND Jolly[i].End>Jolly[i].Start AND
	     Jolly[i].Start<=Sys.Time_CT_DT AND Jolly[i].End>Sys.Time_CT_DT ) THEN
			SetPoint:=Jolly[i].Temp;
	END_IF
END_FOR


(* Status color *)
   IF Alarm   THEN Status_Log:=2; Status_Vis:=COLOR_RED;
ELSIF Warning THEN Status_Log:=1; Status_Vis:=COLOR_YELLOW;
              ELSE Status_Log:=0; Status_Vis:=COLOR_GREEN;
			  END_IF
END_FUNCTION_BLOCK
ACTION DB_Create:
(*
(* Check presence of previous year *)
sFile2:=REPLACE(STR1:=sFile, STR2:=WORD_TO_STRING(Sys.Time_Year-1), L:=4, P:=LEN(FilesPath)+1);
hFile:=SysFileOpen(FileName:=sFile2, Mode:='r');
IF hFile<>0 THEN
	(* Check file version and close *)
	SysFileRead(File:=hFile, Buffer:=ADR(Buf), Size:=1);
	SysFileClose(File:=hFile);
END_IF
IF hFile<>0 AND Buf[0]=1 THEN
	(* Copy file *)
	SysFileCopy(FileDest:=sFile, FileSource:=sFile2);
ELSE
*)
	(* Create empty file *)
	hFile:=SysFileOpen(FileName:=sFile, Mode:='w');

	MEMCLR(pDestinationAddress:=ADR(Buf), BytesToClear:=SIZEOF(Buf));
	FOR i := 0 TO 10239 BY 512 DO
		t1:=SysFileWrite(File:=hFile, Buffer:=ADR(Buf), Size:=512);
	END_FOR
	Buf[0]:=1;
	t2:=SysFileSetPos(File:=hFile, Pos:=0);
	t1:=SysFileWrite(File:=hFile, Buffer:=ADR(Buf), Size:=1);
	SysFileClose(File:=hFile);
(*
END_IF
*)
END_ACTION
ACTION DB_Load:
DB_SetName();

(* Open data file *)
hFile:=SysFileOpen(FileName:=sFile, Mode:='r');

(* File not found *)
IF hFile=0 THEN
	Warning:=TRUE;
	LogEv(EL_Wrn,EO_CRON,ID,1,'No_data_file');
	DB_Create();
	(* Reopen file *)
	hFile:=SysFileOpen(FileName:=sFile, Mode:='r');
	IF hfile=0 THEN
		Alarm:=TRUE;
		LogEv(EL_Alarm,EO_CRON,ID,3,'Filesystem_error');
		RETURN;
	END_IF
END_IF

(* Check version *)
SysFileRead(File:=hFile, Buffer:=ADR(Buf), Size:=1);
IF Buf[0]<>1 THEN
	IF NOT Alarm THEN
		Alarm:=TRUE;
		LogEv(EL_Alarm,EO_CRON,ID,2,'Bad_data_version');
	END_IF
	SysFileClose(File:=hFile);
	RETURN;
END_IF

(* Read Jolly data *)
t2:=SysFileSetPos(File:=hFile, Pos:=512);
t1:=SysFileRead(File:=hFile, Buffer:=ADR(Jolly), Size:=SIZEOF(Jolly));
(* Read active profile index *)
CalendarIdx:=Sys.Time_CT_Day;
t2:=SysFileSetPos(File:=hFile, Pos:=(1024+4*CalendarIdx));
t1:=SysFileRead(File:=hFile, Buffer:=ADR(ProfileNr), Size:=SIZEOF(ProfileNr));
(* Read active profile *)
t2:=SysFileSetPos(File:=hFile, Pos:=(3072+512*ProfileNr));
t1:=SysFileRead(File:=hFile, Buffer:=ADR(Profile), Size:=SIZEOF(Profile));

(* Close file and validate data *)
SysFileClose(File:=hFile);
END_ACTION
ACTION DB_SetName:
(* Create current filename 'yyyyCRnn.DAT' *)
sFile:=CONCAT(FilesPath,WORD_TO_STRING(Sys.Time_Year));
sFile:=CONCAT(STR1:=sFile, STR2:='CR');
IF ID<10 THEN
sFile:=CONCAT(STR1:=sFile, STR2:='0');
END_IF
sFile:=CONCAT(STR1:=sFile, STR2:=BYTE_TO_STRING(ID));
sFile:=CONCAT(STR1:=sFile, STR2:='.DAT');
END_ACTION
ACTION Init:
DB_Load();
InitOK:=TRUE;
END_ACTION

(* POU Plant_Objects/obj_CRON_EDITOR, ST *)
FUNCTION_BLOCK obj_CRON_EDITOR
(* === EDITOR CRONOGRAFO ===
   v1.0[16/04/15] - Versioning
   v1.1[19/05/15] - Create empty profile when not found
*)
VAR_INPUT

	(* Common selections *)
	CN_Sel:			BYTE:=1;
	CN_Act:			BYTE;
	CN_YSel:		WORD:=2015;
	CN_YAct:		WORD;

	(* Profile editor *)
	PR_Sel: 		BYTE:=1;
	PR_Act:			BYTE;
	PR_TT:			REAL;
	PR:				typ_Cron_Profile;
	(* Profile signals *)
	PR_Load:		BOOL;
	PR_Save:		BOOL;

	(* Calendar editor *)
	CA_Sel:			BYTE:=1; (* Calendar month selected *)
	CA_Act:			BYTE;    (* Calendar month active *)
	CA_DayF:		BYTE:=0;
	CA_DayL:		BYTE:=31;
	CA_TPR:			BYTE;
	CA:				typ_Cron_Calendar; (* Only used for first 32 entries *)
	(* Calendar signals *)
	CA_Load:		BOOL;
	CA_Save:		BOOL;

	(* Jolly editor *)
	JL:				ARRAY[0..9] OF typ_Cron_Jolly;
	(* Jolly signals *)
	JL_Load:		BOOL;
	JL_Save:		BOOL;

END_VAR
VAR_OUTPUT
	Message		: STRING;
END_VAR
VAR
	sFileName	: STRING;
	sFileMode	: STRING;
	hFile		: DWORD;
	Buf			: ARRAY[0..512] OF BYTE; (* AVOID THIS!! *)

	i			: WORD;
	ver			: BYTE;
	r1			: BOOL;
	r2			: DWORD;

END_VAR
IF PR_Load THEN PR_Load_Exe(); PR_Load:=FALSE; END_IF
IF PR_Save THEN PR_Save_Exe(); PR_Save:=FALSE; END_IF
IF CA_Load THEN CA_Load_Exe(); CA_Load:=FALSE; END_IF
IF CA_Save THEN CA_Save_Exe(); CA_Save:=FALSE; END_IF
IF JL_Load THEN JL_Load_Exe(); JL_Load:=FALSE; END_IF
IF JL_Save THEN JL_Save_Exe(); JL_Save:=FALSE; END_IF
END_FUNCTION_BLOCK
ACTION CA_Load_Exe:
sFileMode:='r';
FileOpen();

IF hFile<>0 THEN

	(* Read calendar month *)
	FOR i := 0 TO 31 DO
		r1:=SysFileSetPos(File:=hFile, Pos:=(1024 + ((CA_Sel-1)*32 + i)*4));
		r2:=SysFileRead(File:=hFile, Buffer:=ADR(CA.Profile[i]), Size:=1);
	END_FOR

	(* Close file *)
	SysFileClose(File:=hFile);

	(* Validate data *)
	CA_Act :=CA_Sel;
	CN_Act :=CN_Sel;
	CN_YAct:=CN_YSel;

	Message:='Calendar load OK';

END_IF
END_ACTION
ACTION CA_Save_Exe:
sFileMode:='a';
FileOpen();

IF hFile<>0 THEN

	(* Write calendar month *)
	FOR i := 0 TO 31 DO
		r1:=SysFileSetPos(File:=hFile, Pos:=(1024 + ((CA_Sel-1)*32 + i)*4));
		r2:=SysFileGetPos(hFile);
		r2:=SysFileWrite(File:=hFile, Buffer:=ADR(CA.Profile[i]), Size:=1);
	END_FOR

	(* Close file *)
	SysFileClose(File:=hFile);

	Message:='Calendar save OK';

END_IF
END_ACTION
ACTION FileOpen:
(* Create current filename 'yyyyCRnn.DAT' *)
sFileName:=CONCAT(FilesPath,WORD_TO_STRING(CN_YSel));
sFileName:=CONCAT(STR1:=sFileName, STR2:='CR');
IF CN_Sel<10 THEN
sFileName:=CONCAT(STR1:=sFileName, STR2:='0');
END_IF
sFileName:=CONCAT(STR1:=sFileName, STR2:=BYTE_TO_STRING(CN_Sel));
sFileName:=CONCAT(STR1:=sFileName, STR2:='.DAT');

(* Check file version and size! *)
(* ... *)

(* Open data file *)
hFile:=SysFileOpen(FileName:=sFileName, Mode:='r');

(* File not found *)
IF hFile=0 THEN
	Message:='File not found - created empty file';
	(* Create empty file *)
	hFile:=SysFileOpen(FileName:=sFileName, Mode:='w');
	MEMCLR(pDestinationAddress:=ADR(Buf), BytesToClear:=SIZEOF(Buf));
	FOR i := 0 TO 10239 BY 512 DO
		SysFileWrite(File:=hFile, Buffer:=ADR(Buf), Size:=512);
	END_FOR
	Buf[0]:=1;
	SysFileSetPos(File:=hFile, Pos:=0);
	SysFileWrite(File:=hFile, Buffer:=ADR(Buf), Size:=1);
END_IF

(* Close file *)
SysFileClose(File:=hFile);

(* Open data file *)
hFile:=SysFileOpen(FileName:=sFileName, Mode:=sFileMode);
END_ACTION
ACTION JL_Load_Exe:
sFileMode:='r';
FileOpen();

IF hFile<>0 THEN

	(* Read jolly *)
	r1:=SysFileSetPos(File:=hFile, Pos:=512);
	r2:=SysFileRead(File:=hFile, Buffer:=ADR(JL), Size:=SIZEOF(JL));

	(* Close file *)
	SysFileClose(File:=hFile);

	(* Validate data *)
	CN_Act:=CN_Sel;
	CN_YAct:=CN_YSel;

	Message:='Jolly load OK';

END_IF
END_ACTION
ACTION JL_Save_Exe:
sFileMode:='a';
FileOpen();

IF hFile<>0 THEN

	(* Write selected profile *)
	r1:=SysFileSetPos(File:=hFile, Pos:=512);
	r2:=SysFileWrite(File:=hFile, Buffer:=ADR(JL), Size:=SIZEOF(JL));

	(* Close file *)
	SysFileClose(File:=hFile);

	Message:='Jolly save OK';

END_IF
END_ACTION
ACTION PR_Load_Exe:
sFileMode:='r';
FileOpen();

IF hFile<>0 THEN

	(* Read selected profile *)
	r1:=SysFileSetPos(File:=hFile, Pos:=(3072 + 512*PR_Sel));
	r2:=SysFileRead(File:=hFile, Buffer:=ADR(PR), Size:=SIZEOF(PR));

	(* Close file *)
	SysFileClose(File:=hFile);

	(* Validate data *)
	PR_Act:=PR_Sel;
	CN_Act:=CN_Sel;
	CN_YAct:=CN_YSel;

	Message:='Profile load OK';

END_IF
END_ACTION
ACTION PR_Save_Exe:
sFileMode:='a';
FileOpen();

IF hFile<>0 THEN

	(* Write selected profile *)
	r1:=SysFileSetPos(File:=hFile, Pos:=(3072 + 512*PR_Sel));
	r2:=SysFileWrite(File:=hFile, Buffer:=ADR(PR), Size:=SIZEOF(PR));

	(* Close file *)
	SysFileClose(File:=hFile);

	Message:='Profile save OK';

END_IF
END_ACTION

(* POU Plant_Objects/obj_DIFF_ANALOG_IN, ST *)
FUNCTION_BLOCK obj_DIFF_ANALOG_IN
VAR CONSTANT
	NORMAL_STATE:	BYTE := 0;
	LEARN_STATE	:	BYTE := 1;

	SWITCH_ON	:	BYTE := 0;
	READINGS	:	BYTE := 1;
	SWITCH_OFF	:	BYTE := 2;

	LSamples	:	BYTE := 200;	(* Learn samples *)
	MSamples	:	BYTE := 10;		(* Measure samples *)
END_VAR
VAR_INPUT
	ID		:	BYTE;
	Lines   :	BYTE;

	In1		:	BOOL;
	In2		:	BOOL;
	In3		:	BOOL;
	In4		:	BOOL;

	AdcValue:	WORD;
	Tolerance:	WORD;

END_VAR
VAR_OUTPUT

	Out1	:	BOOL;
	Out2	:	BOOL;
	Out3	:	BOOL;
	Out4	:	BOOL;

	OutOfRange	:	BOOL;

END_VAR
VAR
	LearnState	:	BYTE;
	Combination	:	BYTE := 1;
	LSamplesCtr	:	BYTE := 1;
	MSamplesCtr	:	BYTE := 1;
	ActiveLines	:	BYTE;
	Status		:	BYTE;

	ReadValue	:	WORD;
	Threshold_L	:	WORD;
	Threshold_H	:	WORD;

	aLearning	:	ARRAY [1..LSamples] OF WORD;
	aReading	:	ARRAY [1..MSamples] OF WORD;

	SampleTMR	:	TON :=(PT:=T#10ms);
END_VAR
IF Status=NORMAL_STATE THEN
	(* Wait state -> Bypass this block *)
	Out1 := In1;
	Out2 := In2;
	Out3 := In3;
	Out4 := In4;
ELSE
	(* Learning state *)
	Learning();
END_IF
END_FUNCTION_BLOCK
ACTION CheckThreshold:
(* Check actual rele status according to significant rele (line considered in this application) *)
IF Lines = 1 THEN
	ActiveLines.0 := In1;
ELSIF Lines = 2 THEN
		ActiveLines.0 := In1;
		ActiveLines.1 := In2;
ELSIF Lines = 3 THEN
		ActiveLines.0 := In1;
		ActiveLines.1 := In2;
		ActiveLines.2 := In3;
ELSIF Lines = 4 THEN
		ActiveLines.0 := In1;
		ActiveLines.1 := In2;
		ActiveLines.2 := In3;
		ActiveLines.3 := In4;
END_IF

(* Choose the right threshold according to current lines state (switch on or off) *)
IF ActiveLines = 0 THEN
	Threshold_L := 0;
	Threshold_H := (Lux_ref[ID,1] * Tolerance)/100;
ELSE
	Threshold_L := (Lux_ref[ID,ActiveLines] * (100-Tolerance))/100;		(* Low threshold *)
	Threshold_H := (Lux_ref[ID,ActiveLines] * (100+Tolerance))/100;		(* High threshold *)
END_IF

(* Check Alarm *)
IF ReadValue > Threshold_L AND ReadValue < Threshold_H THEN
	OutOfRange := FALSE;
ELSE
	OutOfRange := TRUE;
END_IF
END_ACTION
ACTION Learning:
(* State machine to learn value for each possible combination of lines *)
CASE LearnState OF

	SWITCH_ON:	(* Force switch on of the line and start sampling timer *)

		CASE Combination OF

			1:
				LogEv(EL_Log,EO_SYS,0,4,BYTE_TO_STRING(ID));
				Out1 := TRUE;

			2:
				Out2 := TRUE;

			3:
				Out1 := TRUE;
				Out2 := TRUE;

			4:
				Out3 := TRUE;

			5:
				Out1 := TRUE;
				Out3 := TRUE;

			6:
				Out2 := TRUE;
				Out3 := TRUE;

			7:
				Out1 := TRUE;
				Out2 := TRUE;
				Out3 := TRUE;

			8:
				Out4 := TRUE;

			9:
				Out1 := TRUE;
				Out4 := TRUE;

			10:
				Out2 := TRUE;
				Out4 := TRUE;

			11:
				Out1 := TRUE;
				Out2 := TRUE;
				Out4 := TRUE;

			12:
				Out3 := TRUE;
				Out4 := TRUE;

			13:
				Out1 := TRUE;
				Out3 := TRUE;
				Out4 := TRUE;

			14:
				Out2 := TRUE;
				Out3 := TRUE;
				Out4 := TRUE;

			15:
				Out1 := TRUE;
				Out2 := TRUE;
				Out3 := TRUE;
				Out4 := TRUE;
		END_CASE

		LearnState := READINGS;

	READINGS:	(* Read "SamplesNr" samples, every 10ms *)
		SampleTMR(IN:=NOT SampleTMR.Q);

		IF SampleTMR.Q THEN
			aLearning[LSamplesCtr] := AdcValue;
			LSamplesCtr := LSamplesCtr + 1;

			IF LSamplesCtr = LSamples THEN
				LSamplesCtr := 1;
				SampleTMR(IN:=FALSE);
				LearnState := SWITCH_OFF;
			END_IF
		END_IF

	SWITCH_OFF:	(* Evaluate reference value *)
		CASE Combination OF

			1:
				Out1 := FALSE;

			2:
				Out2 := FALSE;

			3:
				Out1 := FALSE;
				Out2 := FALSE;

			4:
				Out3 := FALSE;

			5:
				Out1 := FALSE;
				Out3 := FALSE;

			6:
				Out2 := FALSE;
				Out3 := FALSE;

			7:
				Out1 := FALSE;
				Out2 := FALSE;
				Out3 := FALSE;

			8:
				Out4 := FALSE;

			9:
				Out1 := FALSE;
				Out4 := FALSE;

			10:
				Out2 := FALSE;
				Out4 := FALSE;

			11:
				Out1 := FALSE;
				Out2 := FALSE;
				Out4 := FALSE;

			12:
				Out3 := FALSE;
				Out4 := FALSE;

			13:
				Out1 := FALSE;
				Out3 := FALSE;
				Out4 := FALSE;

			14:
				Out2 := FALSE;
				Out3 := FALSE;
				Out4 := FALSE;

			15:
				Out1 := FALSE;
				Out2 := FALSE;
				Out3 := FALSE;
				Out4 := FALSE;
		END_CASE

		(* Reference value is the mean value of the measured samples *)
		Lux_ref[ID, Combination] := MEAN_VALUE(ADR(aLearning), LSamples);
		(* Reset readings array *)
		RESET_ARRAY(pData:=ADR(aLearning), Size:=LSamples);

		Combination := Combination + 1;

		IF Combination < EXPT(2,Lines) THEN
			LearnState := SWITCH_ON;
		ELSE
			Combination := 1;
			Status := NORMAL_STATE;			(* Back to wait state *)
			LogEv(EL_Log,EO_SYS,0,5,BYTE_TO_STRING(ID));
		END_IF
END_CASE
END_ACTION
ACTION Measure:
(* Proceed with measure only if not in learning mode *)
IF Status=NORMAL_STATE THEN
	(* If window is full (number of samples as required) go on with mean value e check threshold *)
	IF MSamplesCtr=MSamples THEN

		SHIFT_ARRAY(pData:=ADR(aReading[1]), Size:=MSamples);
		aReading[MSamples] := AdcValue;

		ReadValue := MEAN_VALUE(ADR(aReading), MSamples);
		CheckThreshold();

	ELSE
		(* Window is not full, keep going filling in samples before make a check *)
		aReading[MSamplesCtr] := AdcValue;
		MSamplesCtr := MSamplesCtr + 1;

	END_IF
END_IF
END_ACTION

(* POU Plant_Objects/obj_HVAC_LENNOX_FGK190H2M_new, ST *)
FUNCTION_BLOCK obj_HVAC_LENNOX_FGK190H2M_new
VAR CONSTANT
	Default_SetPointCold	: WORD 	:= 220;
	Default_SetPointHeat	: WORD 	:= 190;
	Default_SetBmsTenv		: INT 	:= -999;
	Default_SetBmsRHenv		: WORD	:= 0;
	Default_SetBmsText		: INT	:= -999;
	Default_SetBmsRHext		: WORD	:= 0;
	Default_MinThrECO		: WORD 	:= 1000;
	Default_MaxThrECO		: WORD 	:= 1500;
END_VAR
VAR_INPUT
	(* Settings *)
	ID						: BYTE;
	ADDRESS					: BYTE:=31;

	(* Controls *)
	Refresh_Period			: TIME:=t#3m;
	Refresh_Auto			: BOOL:=TRUE; (* Enable automatic refresh *)
	Refresh_Now				: BOOL; 	  (* Force an immediate refresh *)

	(* HVAC inputs	*)
	SetPointColdDay			: WORD := 30;	(* Refresh set point	*)
	SetPointHeatDay			: WORD := 30;	(* Heat set point		*)
	SetPointTemp			: WORD;			(* Mean temperature (offset) desired *)

	SetBmsTenv				: INT	:= Default_SetBmsTenv;	(* Environment temperature set point	*)
	SetBmsRHenv				: WORD	:= Default_SetBmsRHenv;	(* Environment humidity set point	*)
	SetBmsText				: INT	:= Default_SetBmsText;	(* External temperature set point 	*)
	SetBmsRHext				: WORD	:= Default_SetBmsRHext;	(* External humidity set point 	*)

	OnOff					: BOOL;

	MinThrECO				: WORD;
	MaxThrECO				: WORD;


	SogliaMinppmCO2				: WORD;
	SogliaMaxppmCO2				: WORD;
	SogliaMinimaSerrandaAria	: WORD;
	TempMinAttFreeCooling		: INT;
	TempMaxAttFreeCooling		: INT;


	WriteBMSGiornoAttivazione : WORD; 			(* ventilatore mandata, bms giorno, set point di attivazione*)
	WriteBMSGiornoAttivazioneZM : WORD;			(* ventilatore mandata, bms giorno, set point di attivazione in zona morta di
															regolazione*)
	WriteBMSNotteAttivazione : WORD; 			(* ventilatore mandata, bms notte, set point di attivazione *)
	WriteBMSNotteAttivazioneZM : WORD;			(* ventilatore mandata, bms notte, set point di attivazione in zona morta di
															regolazione*)


	(* Bit attivazione scrittura parametri in modbus solo se vengono aggiornati *)
	fWriteSP						:BOOL;

	fWriteLimitippmCO2				:BOOL;
	fWriteLimitiSerr				:BOOL;
	fWriteAttivazioneFreeCooling 	:BOOL;
	fWriteAttivazioneSetPoint 		:BOOL;					(* da bilitare mettendo itrue *) 	(*abilitazione scrittura variabile Modbus *)

END_VAR
VAR_IN_OUT
	MODBUS			: obj_MODBUS;
END_VAR
VAR_OUTPUT
	(* Sono read-only tetto il mondo *)
	Data			: typ_MODBUS_HVAC_LENNOX_FGK190H2M_new;
	tmpData			: typ_MODBUS_HVAC_LENNOX_FGK190H2M_new;

	(* Status *)
	Status_Log		: BYTE;
	Status_Vis 		: DWORD;

	ReadSetPointHeatDay			: WORD;
	ReadSetPointColdDay			: WORD;
	ReadSogliaMinimaSerrandaAria: WORD;
	ReadSogliaMinppmCO2			: WORD;
	ReadSogliaMaxppmCO2			: WORD;
	ReadStatoAttivaFreeCooling	: WORD;
	ReadTempMinAttFreeCooling	: INT;   (* valore che può essere negativo *)
	ReadTempMaxAttFreeCooling	: WORD;


	ReadBMSGiornoAttivazione	:WORD;  	(* bms giorno, set point attivazione (86)*)
	ReadBMSGiornoAttivazioneZM	:WORD;  	(* bms giorno, set point attivazione zona morta di regolazione (87) *)
	ReadBMSNotteAttivazione		:WORD;  	(* bms notte, set point attivazione (88) *)
	ReadBMSNotteAttivazioneZM	:WORD;		(* bms notte, set point attivazione zona morta di regolazione (89)*)







END_VAR
VAR
	InitOK		: 	BOOL := FALSE;

	dly 		: 	TON := (PT:=t#5s);
	sta			: 	BYTE; 	(* Status *)
	retry		: 	BYTE;
	fModbusAlr	:	BOOL;

	ModbusAlr	:	FLT_EVENT;
	Alr1		:	FLT_EVENT;
	Alr2		:	FLT_EVENT;
	Alr3		:	FLT_EVENT;
	Alr4		:	FLT_EVENT;
	Alr5		:	FLT_EVENT;
	Alr6		:	FLT_EVENT;
	Alr7		:	FLT_EVENT;

	OldAlarm1	:	WORD;
	OldAlarm2	:	WORD;
	OldAlarm3	:	WORD;
	OldAlarm4	:	WORD;
	OldAlarm5	:	WORD;
	OldAlarm6	:	WORD;
	OldAlarm7	:	WORD;

	ChangedBits	:	WORD;
	AlarmCtr	:	BYTE;

	s1			:	STRING;

	AttivaFreeCooling			: BOOL;
	MacchinaInRaffreddamento	: WORD;
	MacchinaInZonaMorta			: WORD;
	MacchinaInRiscaldamento		: WORD;
	StatoAttivaSwFreeCooling: INT;
END_VAR
Init();

(* Verify inputs are in the right range	*)
CheckInputs();

(* Call ModBus state machine	*)
Stm();

(* Check if an alarm occurs	*)
CheckAlarm();

IF AlarmCtr>0 THEN
	Status_Log 	:= 2;
	Status_Vis	:= COLOR_RED;
ELSE
	Status_Log	:= 0;
	Status_Vis	:= COLOR_GREEN;
END_IF
END_FUNCTION_BLOCK
ACTION AddLogData:
Logger.s1:=INSERT('&HVAC=',BYTE_TO_STRING(ID),5);
IF ID<10 THEN Logger.s1:=INSERT(Logger.s1,'0',5); END_IF

Logger.s1:=CONCAT(Logger.s1,INT_TO_STRING(Data.Tsend));					Logger.s1:=CONCAT(Logger.s1,';');
Logger.s1:=CONCAT(Logger.s1,INT_TO_STRING(Data.Treturn));				Logger.s1:=CONCAT(Logger.s1,';');
Logger.s1:=CONCAT(Logger.s1,WORD_TO_STRING(Data.AirDiffPressure));		Logger.s1:=CONCAT(Logger.s1,';');
Logger.s1:=CONCAT(Logger.s1,WORD_TO_STRING(Data.AirValve));				Logger.s1:=CONCAT(Logger.s1,';');
Logger.s1:=CONCAT(Logger.s1,WORD_TO_STRING(Data.AirGas));				Logger.s1:=CONCAT(Logger.s1,';');
Logger.s1:=CONCAT(Logger.s1,WORD_TO_STRING(Data.Triac));				Logger.s1:=CONCAT(Logger.s1,';');
Logger.s1:=CONCAT(Logger.s1,WORD_TO_STRING(Data.HWB));					Logger.s1:=CONCAT(Logger.s1,';');
Logger.s1:=CONCAT(Logger.s1,WORD_TO_STRING(Data.Humidifier));			Logger.s1:=CONCAT(Logger.s1,';');

(* Create boolean representation of status flag and convert it in string *)
s1:=SEL(Data.StatusFlag.13=TRUE,'0','1');
s1:=CONCAT(s1,SEL(Data.StatusFlag.12=TRUE,'0','1'));
s1:=CONCAT(s1,SEL(Data.StatusFlag.11=TRUE,'0','1'));
s1:=CONCAT(s1,SEL(Data.StatusFlag.10=TRUE,'0','1'));
s1:=CONCAT(s1,SEL(Data.StatusFlag.9=TRUE,'0','1'));
s1:=CONCAT(s1,SEL(Data.StatusFlag.8=TRUE,'0','1'));
s1:=CONCAT(s1,SEL(Data.StatusFlag.7=TRUE,'0','1'));
s1:=CONCAT(s1,SEL(Data.StatusFlag.6=TRUE,'0','1'));
s1:=CONCAT(s1,SEL(Data.StatusFlag.5=TRUE,'0','1'));
s1:=CONCAT(s1,SEL(Data.StatusFlag.4=TRUE,'0','1'));
s1:=CONCAT(s1,SEL(Data.StatusFlag.3=TRUE,'0','1'));
s1:=CONCAT(s1,SEL(Data.StatusFlag.2=TRUE,'0','1'));
s1:=CONCAT(s1,SEL(Data.StatusFlag.1=TRUE,'0','1'));
s1:=CONCAT(s1,SEL(Data.StatusFlag.0=TRUE,'0','1'));

Logger.s1:=CONCAT(Logger.s1,s1);										Logger.s1:=CONCAT(Logger.s1,';');

(* Add operation times *)
Logger.s1:=CONCAT(Logger.s1,DWORD_TO_STRING(Data.HourVent));			Logger.s1:=CONCAT(Logger.s1,';');
Logger.s1:=CONCAT(Logger.s1,DWORD_TO_STRING(Data.HourCir1Comp1));		Logger.s1:=CONCAT(Logger.s1,';');
Logger.s1:=CONCAT(Logger.s1,DWORD_TO_STRING(Data.HourCir1Comp2));		Logger.s1:=CONCAT(Logger.s1,';');
Logger.s1:=CONCAT(Logger.s1,DWORD_TO_STRING(Data.HourCir2Comp1));		Logger.s1:=CONCAT(Logger.s1,';');
Logger.s1:=CONCAT(Logger.s1,DWORD_TO_STRING(Data.HourCir2Comp2));		Logger.s1:=CONCAT(Logger.s1,';');

(* Add actual read SetPoints setted in the HVAC *)
Logger.s1:=CONCAT(Logger.s1,WORD_TO_STRING(ReadSetPointColdDay));			Logger.s1:=CONCAT(Logger.s1,';');
Logger.s1:=CONCAT(Logger.s1,WORD_TO_STRING(Data.ReadSetPointTemp));			Logger.s1:=CONCAT(Logger.s1,';');
Logger.s1:=CONCAT(Logger.s1,WORD_TO_STRING(ReadSetPointHeatDay));			Logger.s1:=CONCAT(Logger.s1,';');

Logger.s1:=CONCAT(Logger.s1,BYTE_TO_STRING(Status_Log));
Logger.s1:=CONCAT(Logger.s1,';');

Logger.s1:=CONCAT(Logger.s1,WORD_TO_STRING(MacchinaInRaffreddamento));
Logger.s1:=CONCAT(Logger.s1,';');
Logger.s1:=CONCAT(Logger.s1,WORD_TO_STRING(MacchinaInZonaMorta));
Logger.s1:=CONCAT(Logger.s1,';');
Logger.s1:=CONCAT(Logger.s1,WORD_TO_STRING(MacchinaInRiscaldamento));
Logger.s1:=CONCAT(Logger.s1,';');

(* Conferma dei valori scritti in modbus *)

Logger.s1:=CONCAT(Logger.s1,WORD_TO_STRING(ReadSogliaMinppmCO2));
Logger.s1:=CONCAT(Logger.s1,';');
Logger.s1:=CONCAT(Logger.s1,WORD_TO_STRING(ReadSogliaMaxppmCO2));
Logger.s1:=CONCAT(Logger.s1,';');
Logger.s1:=CONCAT(Logger.s1,WORD_TO_STRING(ReadSogliaMinimaSerrandaAria));
Logger.s1:=CONCAT(Logger.s1,';');


(* questo bit serve per simulare l' attivazione del free cooling *)
IF Data.Text>ReadTempMinAttFreeCooling AND Data.Text<ReadTempMaxAttFreeCooling THEN
	StatoAttivaSwFreeCooling:=1;  (* Freecooling attivato *)
ELSE
	StatoAttivaSwFreeCooling:=0;  (* Freecooling disattivato *)
END_IF

(* Logger.s1:=CONCAT(Logger.s1,WORD_TO_STRING(ReadStatoAttivaFreeCooling)); *)
Logger.s1:=CONCAT(Logger.s1,INT_TO_STRING(StatoAttivaSwFreeCooling));
Logger.s1:=CONCAT(Logger.s1,';');
Logger.s1:=CONCAT(Logger.s1,WORD_TO_STRING(ReadTempMinAttFreeCooling));
Logger.s1:=CONCAT(Logger.s1,';');
Logger.s1:=CONCAT(Logger.s1,WORD_TO_STRING(ReadTempMaxAttFreeCooling));

Logger.s1:=CONCAT(Logger.s1,';');
Logger.s1:=CONCAT(Logger.s1,INT_TO_STRING(Data.Text));

ADDSTRING(ADR(Logger.TData), ADR(Logger.s1), Logger.TLen);
END_ACTION
ACTION CheckAlarm:
(* Modbus alarm *)
ModbusAlr(IN:=fModbusAlr);

IF ModbusAlr.EVH THEN
	LogEv(EL_Wrn,EO_HVAC,ID,2,SEL(ModBus.MB_MASTER.MB_Error<>0,'0','1'));
	Status_Log := 1;
END_IF

IF ModbusAlr.EVL THEN Status_Log := 0; END_IF	(* If there is an alarm, "Status_Log" wil be overwritten and becomes 2 *)


(***	ALARM 1		***)
(* Verify if at least one bit has changed in register "Alarm 1"	*)
Alr1(IN:=(Data.Alarm1 <> OldAlarm1));

IF Alr1.EVH THEN
	(* Consider just bit(s) that has changed its value (indicated by a logical 1 in "ChangedBits")	*)
	ChangedBits:= Data.Alarm1 XOR OldAlarm1;

	IF ChangedBits.0 THEN
		IF Data.Alarm1.0 THEN LogEv(EL_Alarm,EO_HVAC,ID,3,'70');	AlarmCtr := AlarmCtr + 1;
		ELSE LogEv(EL_Log,EO_HVAC,ID,4,'70'); 						AlarmCtr := AlarmCtr - 1;	END_IF
	END_IF

	IF ChangedBits.1 THEN
		IF Data.Alarm1.1 THEN LogEv(EL_Alarm,EO_HVAC,ID,3,'71');	AlarmCtr := AlarmCtr + 1;
		ELSE LogEv(EL_Log,EO_HVAC,ID,4,'71'); 						AlarmCtr := AlarmCtr - 1;	END_IF
	END_IF

	IF ChangedBits.2 THEN
		IF Data.Alarm1.2 THEN LogEv(EL_Alarm,EO_HVAC,ID,3,'72');	AlarmCtr := AlarmCtr + 1;
		ELSE LogEv(EL_Log,EO_HVAC,ID,4,'72'); 						AlarmCtr := AlarmCtr - 1;	END_IF
	END_IF

	IF ChangedBits.3 THEN
		IF Data.Alarm1.3 THEN LogEv(EL_Alarm,EO_HVAC,ID,3,'9');		AlarmCtr := AlarmCtr + 1;
		ELSE LogEv(EL_Log,EO_HVAC,ID,4,'9'); 						AlarmCtr := AlarmCtr - 1;	END_IF
	END_IF

	IF ChangedBits.4 THEN
		IF Data.Alarm1.4 THEN LogEv(EL_Alarm,EO_HVAC,ID,3,'81');	AlarmCtr := AlarmCtr + 1;
		ELSE LogEv(EL_Log,EO_HVAC,ID,4,'81'); 						AlarmCtr := AlarmCtr - 1;	END_IF
	END_IF

	IF ChangedBits.5 THEN
		IF Data.Alarm1.5 THEN LogEv(EL_Alarm,EO_HVAC,ID,3,'82');	AlarmCtr := AlarmCtr + 1;
		ELSE LogEv(EL_Log,EO_HVAC,ID,4,'82'); 						AlarmCtr := AlarmCtr - 1;	END_IF
	END_IF

	IF ChangedBits.6 THEN
		IF Data.Alarm1.6 THEN LogEv(EL_Alarm,EO_HVAC,ID,3,'83');	AlarmCtr := AlarmCtr + 1;
		ELSE LogEv(EL_Log,EO_HVAC,ID,4,'83'); 						AlarmCtr := AlarmCtr - 1;	END_IF
	END_IF

	IF ChangedBits.7 THEN
		IF Data.Alarm1.7 THEN LogEv(EL_Alarm,EO_HVAC,ID,3,'85');	AlarmCtr := AlarmCtr + 1;
		ELSE LogEv(EL_Log,EO_HVAC,ID,4,'85'); 						AlarmCtr := AlarmCtr - 1;	END_IF
	END_IF

	IF ChangedBits.8 THEN
		IF Data.Alarm1.8 THEN LogEv(EL_Alarm,EO_HVAC,ID,3,'88');	AlarmCtr := AlarmCtr + 1;
		ELSE LogEv(EL_Log,EO_HVAC,ID,4,'88'); 						AlarmCtr := AlarmCtr - 1;	END_IF
	END_IF

	IF ChangedBits.9 THEN
		IF Data.Alarm1.9 THEN LogEv(EL_Alarm,EO_HVAC,ID,3,'22');	AlarmCtr := AlarmCtr + 1;
		ELSE LogEv(EL_Log,EO_HVAC,ID,4,'22'); 						AlarmCtr := AlarmCtr - 1;	END_IF
	END_IF

	IF ChangedBits.10 THEN
		IF Data.Alarm1.10 THEN LogEv(EL_Alarm,EO_HVAC,ID,3,'80');	AlarmCtr := AlarmCtr + 1;
		ELSE LogEv(EL_Log,EO_HVAC,ID,4,'80'); 						AlarmCtr := AlarmCtr - 1;	END_IF
	END_IF

	IF ChangedBits.11 THEN
		IF Data.Alarm1.11 THEN LogEv(EL_Alarm,EO_HVAC,ID,3,'73');	AlarmCtr := AlarmCtr + 1;
		ELSE LogEv(EL_Log,EO_HVAC,ID,4,'73');	 					AlarmCtr := AlarmCtr - 1;	END_IF
	END_IF

	IF ChangedBits.12 THEN
		IF Data.Alarm1.12 THEN LogEv(EL_Alarm,EO_HVAC,ID,3,'1');	AlarmCtr := AlarmCtr + 1;
		ELSE LogEv(EL_Log,EO_HVAC,ID,4,'1'); 						AlarmCtr := AlarmCtr - 1;	END_IF
	END_IF

	IF ChangedBits.13 THEN
		IF Data.Alarm1.13 THEN LogEv(EL_Alarm,EO_HVAC,ID,3,'91');	AlarmCtr := AlarmCtr + 1;
		ELSE LogEv(EL_Log,EO_HVAC,ID,4,'91'); 						AlarmCtr := AlarmCtr - 1;	END_IF
	END_IF

	IF ChangedBits.14 THEN
		IF Data.Alarm1.14 THEN LogEv(EL_Alarm,EO_HVAC,ID,3,'92');	AlarmCtr := AlarmCtr + 1;
		ELSE LogEv(EL_Log,EO_HVAC,ID,4,'92'); 						AlarmCtr := AlarmCtr - 1;	END_IF
	END_IF

	IF ChangedBits.15 THEN
		IF Data.Alarm1.15 THEN LogEv(EL_Alarm,EO_HVAC,ID,3,'99');	AlarmCtr := AlarmCtr + 1;
		ELSE LogEv(EL_Log,EO_HVAC,ID,4,'99'); 						AlarmCtr := AlarmCtr - 1;	END_IF
	END_IF

END_IF


(***	ALARM 2		***)
Alr2(IN:=(Data.Alarm2 <> OldAlarm2));

IF Alr2.EVH THEN

	ChangedBits:= Data.Alarm2 XOR OldAlarm2;

	IF ChangedBits.0 THEN
		IF Data.Alarm2.0 THEN LogEv(EL_Alarm,EO_HVAC,ID,3,'74');	AlarmCtr := AlarmCtr + 1;
		ELSE LogEv(EL_Log,EO_HVAC,ID,4,'74'); 						AlarmCtr := AlarmCtr - 1;	END_IF
	END_IF

	IF ChangedBits.1 THEN
		IF Data.Alarm2.1 THEN LogEv(EL_Alarm,EO_HVAC,ID,3,'93');	AlarmCtr := AlarmCtr + 1;
		ELSE LogEv(EL_Log,EO_HVAC,ID,4,'93'); 						AlarmCtr := AlarmCtr - 1;	END_IF
	END_IF

	IF ChangedBits.2 THEN
		IF Data.Alarm2.2 THEN LogEv(EL_Alarm,EO_HVAC,ID,3,'94');	AlarmCtr := AlarmCtr + 1;
		ELSE LogEv(EL_Log,EO_HVAC,ID,4,'94'); 						AlarmCtr := AlarmCtr - 1;	END_IF
	END_IF

	(* No bit3 for this register	*)

	IF ChangedBits.4 THEN
		IF Data.Alarm2.4 THEN LogEv(EL_Alarm,EO_HVAC,ID,3,'59');	AlarmCtr := AlarmCtr + 1;
		ELSE LogEv(EL_Log,EO_HVAC,ID,4,'59'); 						AlarmCtr := AlarmCtr - 1;	END_IF
	END_IF

	IF ChangedBits.5 THEN
		IF Data.Alarm2.5 THEN LogEv(EL_Alarm,EO_HVAC,ID,3,'56');	AlarmCtr := AlarmCtr + 1;
		ELSE LogEv(EL_Log,EO_HVAC,ID,4,'56'); 						AlarmCtr := AlarmCtr - 1;	END_IF
	END_IF

	IF ChangedBits.6 THEN
		IF Data.Alarm2.6 THEN LogEv(EL_Alarm,EO_HVAC,ID,3,'51');	AlarmCtr := AlarmCtr + 1;
		ELSE LogEv(EL_Log,EO_HVAC,ID,4,'51'); 						AlarmCtr := AlarmCtr - 1;	END_IF
	END_IF

	IF ChangedBits.7 THEN
		IF Data.Alarm2.7 THEN LogEv(EL_Alarm,EO_HVAC,ID,3,'52');	AlarmCtr := AlarmCtr + 1;
		ELSE LogEv(EL_Log,EO_HVAC,ID,4,'52'); 						AlarmCtr := AlarmCtr - 1;	END_IF
	END_IF

	(* No bit8 for this register	*)

	IF ChangedBits.9 THEN
		IF Data.Alarm2.9 THEN LogEv(EL_Alarm,EO_HVAC,ID,3,'13');	AlarmCtr := AlarmCtr + 1;
		ELSE LogEv(EL_Log,EO_HVAC,ID,4,'13'); 						AlarmCtr := AlarmCtr - 1;	END_IF
	END_IF

	IF ChangedBits.10 THEN
		IF Data.Alarm2.10 THEN LogEv(EL_Alarm,EO_HVAC,ID,3,'41');	AlarmCtr := AlarmCtr + 1;
		ELSE LogEv(EL_Log,EO_HVAC,ID,4,'41'); 						AlarmCtr := AlarmCtr - 1;	END_IF
	END_IF

	IF ChangedBits.11 THEN
		IF Data.Alarm2.11 THEN LogEv(EL_Alarm,EO_HVAC,ID,3,'11');	AlarmCtr := AlarmCtr + 1;
		ELSE LogEv(EL_Log,EO_HVAC,ID,4,'11'); 						AlarmCtr := AlarmCtr - 1;	END_IF
	END_IF

	IF ChangedBits.12 THEN
		IF Data.Alarm2.12 THEN LogEv(EL_Alarm,EO_HVAC,ID,3,'12');	AlarmCtr := AlarmCtr + 1;
		ELSE LogEv(EL_Log,EO_HVAC,ID,4,'12'); 						AlarmCtr := AlarmCtr - 1;	END_IF
	END_IF

	IF ChangedBits.13 THEN
		IF Data.Alarm2.13 THEN LogEv(EL_Alarm,EO_HVAC,ID,3,'14');	AlarmCtr := AlarmCtr + 1;
		ELSE LogEv(EL_Log,EO_HVAC,ID,4,'14'); 						AlarmCtr := AlarmCtr - 1;	END_IF
	END_IF

	IF ChangedBits.14 THEN
		IF Data.Alarm2.14 THEN LogEv(EL_Alarm,EO_HVAC,ID,3,'15');	AlarmCtr := AlarmCtr + 1;
		ELSE LogEv(EL_Log,EO_HVAC,ID,4,'15'); 						AlarmCtr := AlarmCtr - 1;	END_IF
	END_IF

	IF ChangedBits.15 THEN
		IF Data.Alarm2.15 THEN LogEv(EL_Alarm,EO_HVAC,ID,3,'16');	AlarmCtr := AlarmCtr + 1;
		ELSE LogEv(EL_Log,EO_HVAC,ID,4,'16'); 						AlarmCtr := AlarmCtr - 1;	END_IF
	END_IF

END_IF


(***	ALARM 3		***)
Alr3(IN:=(Data.Alarm3 <> OldAlarm3));

IF Alr3.EVH THEN

	ChangedBits:= Data.Alarm3 XOR OldAlarm3;

	IF ChangedBits.0 THEN
		IF Data.Alarm3.0 THEN LogEv(EL_Alarm,EO_HVAC,ID,3,'141');	AlarmCtr := AlarmCtr + 1;
		ELSE LogEv(EL_Log,EO_HVAC,ID,4,'141'); 						AlarmCtr := AlarmCtr - 1;	END_IF
	END_IF

	IF ChangedBits.1 THEN
		IF Data.Alarm3.1 THEN LogEv(EL_Alarm,EO_HVAC,ID,3,'142');	AlarmCtr := AlarmCtr + 1;
		ELSE LogEv(EL_Log,EO_HVAC,ID,4,'142'); 						AlarmCtr := AlarmCtr - 1;	END_IF
	END_IF

	IF ChangedBits.2 THEN
		IF Data.Alarm3.2 THEN LogEv(EL_Alarm,EO_HVAC,ID,3,'143');	AlarmCtr := AlarmCtr + 1;
		ELSE LogEv(EL_Log,EO_HVAC,ID,4,'143'); 						AlarmCtr := AlarmCtr - 1;	END_IF
	END_IF

	IF ChangedBits.3 THEN
		IF Data.Alarm3.3 THEN LogEv(EL_Alarm,EO_HVAC,ID,3,'144');	AlarmCtr := AlarmCtr + 1;
		ELSE LogEv(EL_Log,EO_HVAC,ID,4,'144'); 						AlarmCtr := AlarmCtr - 1;	END_IF
	END_IF

	IF ChangedBits.4 THEN
		IF Data.Alarm3.4 THEN LogEv(EL_Alarm,EO_HVAC,ID,3,'114');	AlarmCtr := AlarmCtr + 1;
		ELSE LogEv(EL_Log,EO_HVAC,ID,4,'114'); 						AlarmCtr := AlarmCtr - 1;	END_IF
	END_IF

	IF ChangedBits.5 THEN
		IF Data.Alarm3.5 THEN LogEv(EL_Alarm,EO_HVAC,ID,3,'115');	AlarmCtr := AlarmCtr + 1;
		ELSE LogEv(EL_Log,EO_HVAC,ID,4,'115'); 						AlarmCtr := AlarmCtr - 1;	END_IF
	END_IF

	IF ChangedBits.6 THEN
		IF Data.Alarm3.6 THEN LogEv(EL_Alarm,EO_HVAC,ID,3,'116');	AlarmCtr := AlarmCtr + 1;
		ELSE LogEv(EL_Log,EO_HVAC,ID,4,'116'); 						AlarmCtr := AlarmCtr - 1;	END_IF
	END_IF

	IF ChangedBits.7 THEN
		IF Data.Alarm3.7 THEN LogEv(EL_Alarm,EO_HVAC,ID,3,'117');	AlarmCtr := AlarmCtr + 1;
		ELSE LogEv(EL_Log,EO_HVAC,ID,4,'117'); 						AlarmCtr := AlarmCtr - 1;	END_IF
	END_IF

	IF ChangedBits.8 THEN
		IF Data.Alarm3.8 THEN LogEv(EL_Alarm,EO_HVAC,ID,3,'118');	AlarmCtr := AlarmCtr + 1;
		ELSE LogEv(EL_Log,EO_HVAC,ID,4,'118'); 						AlarmCtr := AlarmCtr - 1;	END_IF
	END_IF

	IF ChangedBits.9 THEN
		IF Data.Alarm3.9 THEN LogEv(EL_Alarm,EO_HVAC,ID,3,'132');	AlarmCtr := AlarmCtr + 1;
		ELSE LogEv(EL_Log,EO_HVAC,ID,4,'132'); 						AlarmCtr := AlarmCtr - 1;	END_IF
	END_IF

	IF ChangedBits.10 THEN
		IF Data.Alarm3.10 THEN LogEv(EL_Alarm,EO_HVAC,ID,3,'75');	AlarmCtr := AlarmCtr + 1;
		ELSE LogEv(EL_Log,EO_HVAC,ID,4,'75'); 						AlarmCtr := AlarmCtr - 1;	END_IF
	END_IF

	IF ChangedBits.11 THEN
		IF Data.Alarm3.11 THEN LogEv(EL_Alarm,EO_HVAC,ID,3,'102');	AlarmCtr := AlarmCtr + 1;
		ELSE LogEv(EL_Log,EO_HVAC,ID,4,'102'); 						AlarmCtr := AlarmCtr - 1;	END_IF
	END_IF

	IF ChangedBits.12 THEN
		IF Data.Alarm3.12 THEN LogEv(EL_Alarm,EO_HVAC,ID,3,'103');	AlarmCtr := AlarmCtr + 1;
		ELSE LogEv(EL_Log,EO_HVAC,ID,4,'103'); 						AlarmCtr := AlarmCtr - 1;	END_IF
	END_IF

	IF ChangedBits.13 THEN
		IF Data.Alarm3.13 THEN LogEv(EL_Alarm,EO_HVAC,ID,3,'86');	AlarmCtr := AlarmCtr + 1;
		ELSE LogEv(EL_Log,EO_HVAC,ID,4,'86'); 						AlarmCtr := AlarmCtr - 1;	END_IF
	END_IF

	IF ChangedBits.14 THEN
		IF Data.Alarm3.14 THEN LogEv(EL_Alarm,EO_HVAC,ID,3,'87');	AlarmCtr := AlarmCtr + 1;
		ELSE LogEv(EL_Log,EO_HVAC,ID,4,'87'); 						AlarmCtr := AlarmCtr - 1;	END_IF
	END_IF

	IF ChangedBits.15 THEN
		IF Data.Alarm3.15 THEN LogEv(EL_Alarm,EO_HVAC,ID,3,'101');	AlarmCtr := AlarmCtr + 1;
		ELSE LogEv(EL_Log,EO_HVAC,ID,4,'101'); 						AlarmCtr := AlarmCtr - 1;	END_IF
	END_IF

END_IF


(***	ALARM 4		***)
Alr4(IN:=(Data.Alarm4 <> OldAlarm4));

IF Alr4.EVH THEN

	ChangedBits:= Data.Alarm4 XOR OldAlarm4;

	IF ChangedBits.0 THEN
		IF Data.Alarm4.0 THEN LogEv(EL_Alarm,EO_HVAC,ID,3,'241');	AlarmCtr := AlarmCtr + 1;
		ELSE LogEv(EL_Log,EO_HVAC,ID,4,'241'); 						AlarmCtr := AlarmCtr - 1;	END_IF
	END_IF

	IF ChangedBits.1 THEN
		IF Data.Alarm4.1 THEN LogEv(EL_Alarm,EO_HVAC,ID,3,'242');	AlarmCtr := AlarmCtr + 1;
		ELSE LogEv(EL_Log,EO_HVAC,ID,4,'242'); 						AlarmCtr := AlarmCtr - 1;	END_IF
	END_IF

	IF ChangedBits.2 THEN
		IF Data.Alarm4.2 THEN LogEv(EL_Alarm,EO_HVAC,ID,3,'243');	AlarmCtr := AlarmCtr + 1;
		ELSE LogEv(EL_Log,EO_HVAC,ID,4,'243'); 						AlarmCtr := AlarmCtr - 1;	END_IF
	END_IF

	IF ChangedBits.3 THEN
		IF Data.Alarm4.3 THEN LogEv(EL_Alarm,EO_HVAC,ID,3,'244');	AlarmCtr := AlarmCtr + 1;
		ELSE LogEv(EL_Log,EO_HVAC,ID,4,'244'); 						AlarmCtr := AlarmCtr - 1;	END_IF
	END_IF

	IF ChangedBits.4 THEN
		IF Data.Alarm4.4 THEN LogEv(EL_Alarm,EO_HVAC,ID,3,'214');	AlarmCtr := AlarmCtr + 1;
		ELSE LogEv(EL_Log,EO_HVAC,ID,4,'214'); 						AlarmCtr := AlarmCtr - 1;	END_IF
	END_IF

	IF ChangedBits.5 THEN
		IF Data.Alarm4.5 THEN LogEv(EL_Alarm,EO_HVAC,ID,3,'215');	AlarmCtr := AlarmCtr + 1;
		ELSE LogEv(EL_Log,EO_HVAC,ID,4,'215'); 						AlarmCtr := AlarmCtr - 1;	END_IF
	END_IF

	IF ChangedBits.6 THEN
		IF Data.Alarm4.6 THEN LogEv(EL_Alarm,EO_HVAC,ID,3,'216');	AlarmCtr := AlarmCtr + 1;
		ELSE LogEv(EL_Log,EO_HVAC,ID,4,'216'); 						AlarmCtr := AlarmCtr - 1;	END_IF
	END_IF

	IF ChangedBits.7 THEN
		IF Data.Alarm4.7 THEN LogEv(EL_Alarm,EO_HVAC,ID,3,'217');	AlarmCtr := AlarmCtr + 1;
		ELSE LogEv(EL_Log,EO_HVAC,ID,4,'217'); 						AlarmCtr := AlarmCtr - 1;	END_IF
	END_IF

	IF ChangedBits.8 THEN
		IF Data.Alarm4.8 THEN LogEv(EL_Alarm,EO_HVAC,ID,3,'218');	AlarmCtr := AlarmCtr + 1;
		ELSE LogEv(EL_Log,EO_HVAC,ID,4,'218'); 						AlarmCtr := AlarmCtr - 1;	END_IF
	END_IF

	IF ChangedBits.9 THEN
		IF Data.Alarm4.9 THEN LogEv(EL_Alarm,EO_HVAC,ID,3,'232');	AlarmCtr := AlarmCtr + 1;
		ELSE LogEv(EL_Log,EO_HVAC,ID,4,'232'); 						AlarmCtr := AlarmCtr - 1;	END_IF
	END_IF

	IF ChangedBits.10 THEN
		IF Data.Alarm4.10 THEN LogEv(EL_Alarm,EO_HVAC,ID,3,'76');	AlarmCtr := AlarmCtr + 1;
		ELSE LogEv(EL_Log,EO_HVAC,ID,4,'76'); 						AlarmCtr := AlarmCtr - 1;	END_IF
	END_IF

	IF ChangedBits.11 THEN
		IF Data.Alarm4.11 THEN LogEv(EL_Alarm,EO_HVAC,ID,3,'202');	AlarmCtr := AlarmCtr + 1;
		ELSE LogEv(EL_Log,EO_HVAC,ID,4,'202'); 						AlarmCtr := AlarmCtr - 1;	END_IF
	END_IF

	IF ChangedBits.12 THEN
		IF Data.Alarm4.12 THEN LogEv(EL_Alarm,EO_HVAC,ID,3,'203');	AlarmCtr := AlarmCtr + 1;
		ELSE LogEv(EL_Log,EO_HVAC,ID,4,'203'); 						AlarmCtr := AlarmCtr - 1;	END_IF
	END_IF

	IF ChangedBits.13 THEN
		IF Data.Alarm4.13 THEN LogEv(EL_Alarm,EO_HVAC,ID,3,'2');	AlarmCtr := AlarmCtr + 1;
		ELSE LogEv(EL_Log,EO_HVAC,ID,4,'2'); 						AlarmCtr := AlarmCtr - 1;	END_IF
	END_IF

	IF ChangedBits.14 THEN
		IF Data.Alarm4.14 THEN LogEv(EL_Alarm,EO_HVAC,ID,3,'25');	AlarmCtr := AlarmCtr + 1;
		ELSE LogEv(EL_Log,EO_HVAC,ID,4,'25'); 						AlarmCtr := AlarmCtr - 1;	END_IF
	END_IF

	IF ChangedBits.15 THEN
		IF Data.Alarm4.15 THEN LogEv(EL_Alarm,EO_HVAC,ID,3,'26');	AlarmCtr := AlarmCtr + 1;
		ELSE LogEv(EL_Log,EO_HVAC,ID,4,'26'); 						AlarmCtr := AlarmCtr - 1;	END_IF
	END_IF

END_IF


(***	ALARM 5		***)
Alr5(IN:=(Data.Alarm5 <> OldAlarm5));

IF Alr5.EVH THEN

	ChangedBits:= Data.Alarm5 XOR OldAlarm5;

	IF ChangedBits.0 THEN
		IF Data.Alarm5.0 THEN LogEv(EL_Alarm,EO_HVAC,ID,3,'84');	AlarmCtr := AlarmCtr + 1;
		ELSE LogEv(EL_Log,EO_HVAC,ID,4,'84'); 						AlarmCtr := AlarmCtr - 1;	END_IF
	END_IF

	IF ChangedBits.1 THEN
		IF Data.Alarm5.1 THEN LogEv(EL_Alarm,EO_HVAC,ID,3,'23');	AlarmCtr := AlarmCtr + 1;
		ELSE LogEv(EL_Log,EO_HVAC,ID,4,'23'); 						AlarmCtr := AlarmCtr - 1;	END_IF
	END_IF

	IF ChangedBits.2 THEN
		IF Data.Alarm5.2 THEN LogEv(EL_Alarm,EO_HVAC,ID,3,'24');	AlarmCtr := AlarmCtr + 1;
		ELSE LogEv(EL_Log,EO_HVAC,ID,4,'24'); 						AlarmCtr := AlarmCtr - 1;	END_IF
	END_IF

	IF ChangedBits.3 THEN
		IF Data.Alarm5.3 THEN LogEv(EL_Alarm,EO_HVAC,ID,3,'32');	AlarmCtr := AlarmCtr + 1;
		ELSE LogEv(EL_Log,EO_HVAC,ID,4,'32'); 						AlarmCtr := AlarmCtr - 1;	END_IF
	END_IF

	IF ChangedBits.4 THEN
		IF Data.Alarm5.4 THEN LogEv(EL_Alarm,EO_HVAC,ID,3,'33');	AlarmCtr := AlarmCtr + 1;
		ELSE LogEv(EL_Log,EO_HVAC,ID,4,'33'); 						AlarmCtr := AlarmCtr - 1;	END_IF
	END_IF

	IF ChangedBits.5 THEN
		IF Data.Alarm5.5 THEN LogEv(EL_Alarm,EO_HVAC,ID,3,'21');	AlarmCtr := AlarmCtr + 1;
		ELSE LogEv(EL_Log,EO_HVAC,ID,4,'21'); 						AlarmCtr := AlarmCtr - 1;	END_IF
	END_IF

	IF ChangedBits.6 THEN
		IF Data.Alarm5.6 THEN LogEv(EL_Alarm,EO_HVAC,ID,3,'4');		AlarmCtr := AlarmCtr + 1;
		ELSE LogEv(EL_Log,EO_HVAC,ID,4,'4'); 						AlarmCtr := AlarmCtr - 1;	END_IF
	END_IF

	IF ChangedBits.7 THEN
		IF Data.Alarm5.7 THEN LogEv(EL_Alarm,EO_HVAC,ID,3,'5');		AlarmCtr := AlarmCtr + 1;
		ELSE LogEv(EL_Log,EO_HVAC,ID,4,'5'); 						AlarmCtr := AlarmCtr - 1;	END_IF
	END_IF

	IF ChangedBits.8 THEN
		IF Data.Alarm5.8 THEN LogEv(EL_Alarm,EO_HVAC,ID,3,'89');	AlarmCtr := AlarmCtr + 1;
		ELSE LogEv(EL_Log,EO_HVAC,ID,4,'89'); 						AlarmCtr := AlarmCtr - 1;	END_IF
	END_IF

	IF ChangedBits.9 THEN
		IF Data.Alarm5.9 THEN LogEv(EL_Alarm,EO_HVAC,ID,3,'29');	AlarmCtr := AlarmCtr + 1;
		ELSE LogEv(EL_Log,EO_HVAC,ID,4,'29'); 						AlarmCtr := AlarmCtr - 1;	END_IF
	END_IF

	IF ChangedBits.10 THEN
		IF Data.Alarm5.10 THEN LogEv(EL_Alarm,EO_HVAC,ID,3,'54');	AlarmCtr := AlarmCtr + 1;
		ELSE LogEv(EL_Log,EO_HVAC,ID,4,'54'); 						AlarmCtr := AlarmCtr - 1;	END_IF
	END_IF

	IF ChangedBits.11 THEN
		IF Data.Alarm5.11 THEN LogEv(EL_Alarm,EO_HVAC,ID,3,'31');	AlarmCtr := AlarmCtr + 1;
		ELSE LogEv(EL_Log,EO_HVAC,ID,4,'31'); 						AlarmCtr := AlarmCtr - 1;	END_IF
	END_IF

	(* No bit12 and bit13 for this register	*)

	IF ChangedBits.14 THEN
		IF Data.Alarm5.14 THEN LogEv(EL_Alarm,EO_HVAC,ID,3,'110');	AlarmCtr := AlarmCtr + 1;
		ELSE LogEv(EL_Log,EO_HVAC,ID,4,'110'); 						AlarmCtr := AlarmCtr - 1;	END_IF
	END_IF

	IF ChangedBits.15 THEN
		IF Data.Alarm5.15 THEN LogEv(EL_Alarm,EO_HVAC,ID,3,'210');	AlarmCtr := AlarmCtr + 1;
		ELSE LogEv(EL_Log,EO_HVAC,ID,4,'210'); 						AlarmCtr := AlarmCtr - 1;	END_IF
	END_IF

END_IF


(***	ALARM 6		***)
Alr6(IN:=(Data.Alarm6 <> OldAlarm6));

IF Alr6.EVH THEN

	ChangedBits:= Data.Alarm6 XOR OldAlarm6;

	IF ChangedBits.0 THEN
		IF Data.Alarm6.0 THEN LogEv(EL_Alarm,EO_HVAC,ID,3,'119');	AlarmCtr := AlarmCtr + 1;
		ELSE LogEv(EL_Log,EO_HVAC,ID,4,'119'); 						AlarmCtr := AlarmCtr - 1;	END_IF
	END_IF

	IF ChangedBits.1 THEN
		IF Data.Alarm6.1 THEN LogEv(EL_Alarm,EO_HVAC,ID,3,'129');	AlarmCtr := AlarmCtr + 1;
		ELSE LogEv(EL_Log,EO_HVAC,ID,4,'129');	 					AlarmCtr := AlarmCtr - 1;	END_IF
	END_IF

	IF ChangedBits.2 THEN
		IF Data.Alarm6.2 THEN LogEv(EL_Alarm,EO_HVAC,ID,3,'128');	AlarmCtr := AlarmCtr + 1;
		ELSE LogEv(EL_Log,EO_HVAC,ID,4,'128'); 						AlarmCtr := AlarmCtr - 1;	END_IF
	END_IF

	IF ChangedBits.3 THEN
		IF Data.Alarm6.3 THEN LogEv(EL_Alarm,EO_HVAC,ID,3,'127');	AlarmCtr := AlarmCtr + 1;
		ELSE LogEv(EL_Log,EO_HVAC,ID,4,'127'); 						AlarmCtr := AlarmCtr - 1;	END_IF
	END_IF

	IF ChangedBits.4 THEN
		IF Data.Alarm6.4 THEN LogEv(EL_Alarm,EO_HVAC,ID,3,'121');	AlarmCtr := AlarmCtr + 1;
		ELSE LogEv(EL_Log,EO_HVAC,ID,4,'121'); 						AlarmCtr := AlarmCtr - 1;	END_IF
	END_IF

	IF ChangedBits.5 THEN
		IF Data.Alarm6.5 THEN LogEv(EL_Alarm,EO_HVAC,ID,3,'122');	AlarmCtr := AlarmCtr + 1;
		ELSE LogEv(EL_Log,EO_HVAC,ID,4,'122'); 						AlarmCtr := AlarmCtr - 1;	END_IF
	END_IF

	IF ChangedBits.6 THEN
		IF Data.Alarm6.6 THEN LogEv(EL_Alarm,EO_HVAC,ID,3,'123');	AlarmCtr := AlarmCtr + 1;
		ELSE LogEv(EL_Log,EO_HVAC,ID,4,'123'); 						AlarmCtr := AlarmCtr - 1;	END_IF
	END_IF

	IF ChangedBits.7 THEN
		IF Data.Alarm6.7 THEN LogEv(EL_Alarm,EO_HVAC,ID,3,'124');	AlarmCtr := AlarmCtr + 1;
		ELSE LogEv(EL_Log,EO_HVAC,ID,4,'124'); 						AlarmCtr := AlarmCtr - 1;	END_IF
	END_IF

	IF ChangedBits.8 THEN
		IF Data.Alarm6.8 THEN LogEv(EL_Alarm,EO_HVAC,ID,3,'219');	AlarmCtr := AlarmCtr + 1;
		ELSE LogEv(EL_Log,EO_HVAC,ID,4,'219'); 						AlarmCtr := AlarmCtr - 1;	END_IF
	END_IF

	IF ChangedBits.9 THEN
		IF Data.Alarm6.9 THEN LogEv(EL_Alarm,EO_HVAC,ID,3,'229');	AlarmCtr := AlarmCtr + 1;
		ELSE LogEv(EL_Log,EO_HVAC,ID,4,'229'); 						AlarmCtr := AlarmCtr - 1;	END_IF
	END_IF

	IF ChangedBits.10 THEN
		IF Data.Alarm6.10 THEN LogEv(EL_Alarm,EO_HVAC,ID,3,'228');	AlarmCtr := AlarmCtr + 1;
		ELSE LogEv(EL_Log,EO_HVAC,ID,4,'228'); 						AlarmCtr := AlarmCtr - 1;	END_IF
	END_IF

	IF ChangedBits.11 THEN
		IF Data.Alarm6.11 THEN LogEv(EL_Alarm,EO_HVAC,ID,3,'227');	AlarmCtr := AlarmCtr + 1;
		ELSE LogEv(EL_Log,EO_HVAC,ID,4,'227'); 						AlarmCtr := AlarmCtr - 1;	END_IF
	END_IF

	IF ChangedBits.12 THEN
		IF Data.Alarm6.12 THEN LogEv(EL_Alarm,EO_HVAC,ID,3,'221');	AlarmCtr := AlarmCtr + 1;
		ELSE LogEv(EL_Log,EO_HVAC,ID,4,'221'); 						AlarmCtr := AlarmCtr - 1;	END_IF
	END_IF

	IF ChangedBits.13 THEN
		IF Data.Alarm6.13 THEN LogEv(EL_Alarm,EO_HVAC,ID,3,'222');	AlarmCtr := AlarmCtr + 1;
		ELSE LogEv(EL_Log,EO_HVAC,ID,4,'222');	 					AlarmCtr := AlarmCtr - 1;	END_IF
	END_IF

	IF ChangedBits.14 THEN
		IF Data.Alarm6.14 THEN LogEv(EL_Alarm,EO_HVAC,ID,3,'223');	AlarmCtr := AlarmCtr + 1;
		ELSE LogEv(EL_Log,EO_HVAC,ID,4,'223'); 						AlarmCtr := AlarmCtr - 1;	END_IF
	END_IF

	IF ChangedBits.15 THEN
		IF Data.Alarm6.15 THEN LogEv(EL_Alarm,EO_HVAC,ID,3,'224');	AlarmCtr := AlarmCtr + 1;
		ELSE LogEv(EL_Log,EO_HVAC,ID,4,'224'); 						AlarmCtr := AlarmCtr - 1;	END_IF
	END_IF

END_IF


(***	ALARM 7		***)
Alr7(IN:=(Data.Alarm7 <> OldAlarm7));

IF Alr7.EVH THEN

	ChangedBits:= Data.Alarm7 XOR OldAlarm7;

	IF ChangedBits.0 THEN
		IF Data.Alarm7.0 THEN LogEv(EL_Alarm,EO_HVAC,ID,3,'341');	AlarmCtr := AlarmCtr + 1;
		ELSE LogEv(EL_Log,EO_HVAC,ID,4,'341'); 						AlarmCtr := AlarmCtr - 1;	END_IF
	END_IF

	IF ChangedBits.1 THEN
		IF Data.Alarm7.1 THEN LogEv(EL_Alarm,EO_HVAC,ID,3,'342');	AlarmCtr := AlarmCtr + 1;
		ELSE LogEv(EL_Log,EO_HVAC,ID,4,'342'); 						AlarmCtr := AlarmCtr - 1;	END_IF
	END_IF

	IF ChangedBits.2 THEN
		IF Data.Alarm7.2 THEN LogEv(EL_Alarm,EO_HVAC,ID,3,'343');	AlarmCtr := AlarmCtr + 1;
		ELSE LogEv(EL_Log,EO_HVAC,ID,4,'343'); 						AlarmCtr := AlarmCtr - 1;	END_IF
	END_IF

	IF ChangedBits.3 THEN
		IF Data.Alarm7.3 THEN LogEv(EL_Alarm,EO_HVAC,ID,3,'344');	AlarmCtr := AlarmCtr + 1;
		ELSE LogEv(EL_Log,EO_HVAC,ID,4,'344'); 						AlarmCtr := AlarmCtr - 1;	END_IF
	END_IF

	IF ChangedBits.4 THEN
		IF Data.Alarm7.4 THEN LogEv(EL_Alarm,EO_HVAC,ID,3,'314');	AlarmCtr := AlarmCtr + 1;
		ELSE LogEv(EL_Log,EO_HVAC,ID,4,'314'); 						AlarmCtr := AlarmCtr - 1;	END_IF
	END_IF

	IF ChangedBits.5 THEN
		IF Data.Alarm7.5 THEN LogEv(EL_Alarm,EO_HVAC,ID,3,'315');	AlarmCtr := AlarmCtr + 1;
		ELSE LogEv(EL_Log,EO_HVAC,ID,4,'315'); 						AlarmCtr := AlarmCtr - 1;	END_IF
	END_IF

	IF ChangedBits.6 THEN
		IF Data.Alarm7.6 THEN LogEv(EL_Alarm,EO_HVAC,ID,3,'316');	AlarmCtr := AlarmCtr + 1;
		ELSE LogEv(EL_Log,EO_HVAC,ID,4,'316'); 						AlarmCtr := AlarmCtr - 1;	END_IF
	END_IF

	IF ChangedBits.7 THEN
		IF Data.Alarm7.7 THEN LogEv(EL_Alarm,EO_HVAC,ID,3,'317');	AlarmCtr := AlarmCtr + 1;
		ELSE LogEv(EL_Log,EO_HVAC,ID,4,'317'); 						AlarmCtr := AlarmCtr - 1;	END_IF
	END_IF

	IF ChangedBits.8 THEN
		IF Data.Alarm7.8 THEN LogEv(EL_Alarm,EO_HVAC,ID,3,'319');	AlarmCtr := AlarmCtr + 1;
		ELSE LogEv(EL_Log,EO_HVAC,ID,4,'319'); 						AlarmCtr := AlarmCtr - 1;	END_IF
	END_IF

	IF ChangedBits.9 THEN
		IF Data.Alarm7.9 THEN LogEv(EL_Alarm,EO_HVAC,ID,3,'329');	AlarmCtr := AlarmCtr + 1;
		ELSE LogEv(EL_Log,EO_HVAC,ID,4,'329'); 						AlarmCtr := AlarmCtr - 1;	END_IF
	END_IF

	IF ChangedBits.10 THEN
		IF Data.Alarm7.10 THEN LogEv(EL_Alarm,EO_HVAC,ID,3,'328');	AlarmCtr := AlarmCtr + 1;
		ELSE LogEv(EL_Log,EO_HVAC,ID,4,'328'); 						AlarmCtr := AlarmCtr - 1;	END_IF
	END_IF

	IF ChangedBits.11 THEN
		IF Data.Alarm7.11 THEN LogEv(EL_Alarm,EO_HVAC,ID,3,'327');	AlarmCtr := AlarmCtr + 1;
		ELSE LogEv(EL_Log,EO_HVAC,ID,4,'327'); 						AlarmCtr := AlarmCtr - 1;	END_IF
	END_IF

	IF ChangedBits.12 THEN
		IF Data.Alarm7.12 THEN LogEv(EL_Alarm,EO_HVAC,ID,3,'321');	AlarmCtr := AlarmCtr + 1;
		ELSE LogEv(EL_Log,EO_HVAC,ID,4,'321'); 						AlarmCtr := AlarmCtr - 1;	END_IF
	END_IF

	IF ChangedBits.13 THEN
		IF Data.Alarm7.13 THEN LogEv(EL_Alarm,EO_HVAC,ID,3,'322');	AlarmCtr := AlarmCtr + 1;
		ELSE LogEv(EL_Log,EO_HVAC,ID,4,'322'); 						AlarmCtr := AlarmCtr - 1;	END_IF
	END_IF

	IF ChangedBits.14 THEN
		IF Data.Alarm7.14 THEN LogEv(EL_Alarm,EO_HVAC,ID,3,'323');	AlarmCtr := AlarmCtr + 1;
		ELSE LogEv(EL_Log,EO_HVAC,ID,4,'323'); 						AlarmCtr := AlarmCtr - 1;	END_IF
	END_IF

	IF ChangedBits.15 THEN
		IF Data.Alarm7.15 THEN LogEv(EL_Alarm,EO_HVAC,ID,3,'324');	AlarmCtr := AlarmCtr + 1;
		ELSE LogEv(EL_Log,EO_HVAC,ID,4,'324'); 						AlarmCtr := AlarmCtr - 1;	END_IF
	END_IF

END_IF
END_ACTION
ACTION CheckInputs:
(* If value of variables are out of admissible range, set default value as stated in the manual	*)


(* nuova gestione di queste variabili
IF SetPointColdDay<80 OR SetPointColdDay>350 THEN SetPointColdDay := Default_SetPointCold; END_IF
IF SetPointHeatDay<80 OR SetPointHeatDay>350 THEN SetPointHeatDay := Default_SetPointHeat; END_IF
*)
IF SetBmsTenv<-999 OR SetBmsTenv>999 THEN SetBmsTenv := Default_SetBmsTenv; END_IF
IF SetBmsRHenv<0 OR SetBmsRHenv>1000 THEN SetBmsRHenv := Default_SetBmsRHenv; END_IF
IF SetBmsText<-999 OR SetBmsText>999 THEN SetBmsText := Default_SetBmsText; END_IF
IF SetBmsRHext<0 OR SetBmsRHext>1000 THEN SetBmsRHext := Default_SetBmsRHext; END_IF

IF MinThrECO<0 OR MinThrECO>2000 THEN MinThrECO := Default_MinThrECO; END_IF
IF MaxThrECO<0 OR MaxThrECO>2000 THEN MaxThrECO := Default_MaxThrECO; END_IF
END_ACTION
ACTION Init:
IF NOT InitOK THEN

	fWriteSP := TRUE;
	InitOK := TRUE;

END_IF
END_ACTION
ACTION Stm:
CASE sta OF
	0: (* === Wait update signals *)
		dly(IN:=NOT (dly.Q OR Refresh_Now OR (NOT Refresh_Auto)));
		IF dly.Q OR Refresh_Now THEN
			dly.PT := Refresh_Period;
			Refresh_Now := FALSE;

			retry := 0;
			sta := 1;
		END_IF

	1: (* === Start update when MB is free *)
		IF NOT (MODBUS.MB_Lock OR MODBUS.MB_Start) THEN

			MODBUS.MB_Lock := TRUE;

			MODBUS.MB_Query.SlaveAddress		:= ADDRESS;
			MODBUS.MB_Query.FunctionCode		:= 16#03;
			MODBUS.MB_Query.Read_StartAddress	:= 36;
			MODBUS.MB_Query.Read_Quantity		:= 16;

			MODBUS.MB_Start := TRUE;
			sta := 2;
		END_IF

	2:	(* Lettura Varibili dal campo - Segnali Vari *)
		IF NOT MODBUS.MB_Start THEN
			IF MODBUS.MB_MASTER.MB_Error<>MB_NO_ERROR OR MODBUS.MB_Resp.Error<>0 THEN
				sta:=100;
			ELSE

				tmpData.AlarmCode			:= MODBUS.MB_Resp.Data[0];
				tmpData.Tenv				:= WORD_TO_INT(MODBUS.MB_Resp.Data[1]);
				tmpData.Text				:= WORD_TO_INT(MODBUS.MB_Resp.Data[2]);
				tmpData.Tsend				:= WORD_TO_INT(MODBUS.MB_Resp.Data[3]);
				tmpData.Treturn				:= WORD_TO_INT(MODBUS.MB_Resp.Data[4]);
				tmpData.RH_env				:= MODBUS.MB_Resp.Data[5];
				tmpData.AH_env				:= MODBUS.MB_Resp.Data[6];
				tmpData.RH_ext				:= MODBUS.MB_Resp.Data[7];
				tmpData.AH_ext				:= MODBUS.MB_Resp.Data[8];
				tmpData.AirDiffPressure		:= MODBUS.MB_Resp.Data[9];
				tmpData.CO2_ppm				:= MODBUS.MB_Resp.Data[10];
				tmpData.AirValve			:= MODBUS.MB_Resp.Data[11];
				tmpData.AirGas				:= MODBUS.MB_Resp.Data[12];
				tmpData.Triac				:= MODBUS.MB_Resp.Data[13];
				tmpData.HWB					:= MODBUS.MB_Resp.Data[14];
				tmpData.Humidifier			:= MODBUS.MB_Resp.Data[15];

				MODBUS.MB_Query.SlaveAddress		:= ADDRESS;
				MODBUS.MB_Query.FunctionCode		:= 16#03;
				MODBUS.MB_Query.Read_StartAddress	:= 62;
				MODBUS.MB_Query.Read_Quantity		:= 10;

				MODBUS.MB_Start := TRUE;
				sta := 3;

			END_IF
		END_IF

	3:	(* Stato contatori h per segnalazione lavoro *)
		IF NOT MODBUS.MB_Start THEN
			IF MODBUS.MB_MASTER.MB_Error<>MB_NO_ERROR OR MODBUS.MB_Resp.Error<>0 THEN
				sta:=100;
			ELSE

				tmpData.HourVent 		:= BUILD_16TO32(ADR(MODBUS.MB_Resp.Data[0]));
				tmpData.HourCir1Comp1 	:= BUILD_16TO32(ADR(MODBUS.MB_Resp.Data[2]));
				tmpData.HourCir1Comp2 	:= BUILD_16TO32(ADR(MODBUS.MB_Resp.Data[4]));
				tmpData.HourCir2Comp1 	:= BUILD_16TO32(ADR(MODBUS.MB_Resp.Data[6]));
				tmpData.HourCir2Comp2	:= BUILD_16TO32(ADR(MODBUS.MB_Resp.Data[8]));

				MODBUS.MB_Query.SlaveAddress		:= ADDRESS;
				MODBUS.MB_Query.FunctionCode		:= 16#03;
				MODBUS.MB_Query.Read_StartAddress	:= 74;
				MODBUS.MB_Query.Read_Quantity		:= 7;

				MODBUS.MB_Start := TRUE;
				sta := 4;

			END_IF
		END_IF

	4:	(* lettura allarmi attivi  *)
		IF NOT MODBUS.MB_Start THEN
			IF MODBUS.MB_MASTER.MB_Error<>MB_NO_ERROR OR MODBUS.MB_Resp.Error<>0 THEN
				sta:=100;
			ELSE
				tmpData.Alarm1	:= MODBUS.MB_Resp.Data[0];
				tmpData.Alarm2	:= MODBUS.MB_Resp.Data[1];
				tmpData.Alarm3	:= MODBUS.MB_Resp.Data[2];
				tmpData.Alarm4	:= MODBUS.MB_Resp.Data[3];
				tmpData.Alarm5	:= MODBUS.MB_Resp.Data[4];
				tmpData.Alarm6	:= MODBUS.MB_Resp.Data[5];
				tmpData.Alarm7	:= MODBUS.MB_Resp.Data[6];

				(*MODBUS.MB_Query.SlaveAddress		:= ADDRESS;
				MODBUS.MB_Query.FunctionCode		:= 16#03;
				MODBUS.MB_Query.Read_StartAddress	:= 134;
				MODBUS.MB_Query.Read_Quantity		:= 16;*)
				MODBUS.MB_Query.SlaveAddress		:= ADDRESS;
				MODBUS.MB_Query.FunctionCode		:= 16#03;
				MODBUS.MB_Query.Read_StartAddress	:= 33;
				MODBUS.MB_Query.Read_Quantity		:= 3;


				MODBUS.MB_Start := TRUE;
				sta := 5;
			END_IF
		END_IF

	5:  (* Set Point attivi *)
		IF NOT MODBUS.MB_Start THEN
			IF MODBUS.MB_MASTER.MB_Error<>MB_NO_ERROR OR MODBUS.MB_Resp.Error<>0 THEN
				sta:=100;
			ELSE
				tmpData.ReadSetPointCold :=  MODBUS.MB_Resp.Data[0];
				tmpData.ReadSetPointTemp :=  MODBUS.MB_Resp.Data[1];
				tmpData.ReadSetPointHeat :=  MODBUS.MB_Resp.Data[2];

				MODBUS.MB_Query.SlaveAddress		:= ADDRESS;
				MODBUS.MB_Query.FunctionCode		:= 16#03;
				MODBUS.MB_Query.Read_StartAddress	:= 134;
				MODBUS.MB_Query.Read_Quantity		:= 16;

				MODBUS.MB_Start := TRUE;
				sta := 10;
			END_IF
		END_IF

	(* 	WRITE	*)

	10:	(* Write parametro watch dog HVAC	*)
		IF NOT MODBUS.MB_Start THEN
			IF MODBUS.MB_MASTER.MB_Error<>MB_NO_ERROR OR MODBUS.MB_Resp.Error<>0 THEN
				sta:=100;
			ELSE
				tmpData.StatusFlag.0 := WORD_TO_BOOL(MODBUS.MB_Resp.Data[0]);
				tmpData.StatusFlag.1 := WORD_TO_BOOL(MODBUS.MB_Resp.Data[1]);
				tmpData.StatusFlag.2 := WORD_TO_BOOL(MODBUS.MB_Resp.Data[2]);
				tmpData.StatusFlag.3 := WORD_TO_BOOL(MODBUS.MB_Resp.Data[3]);
				tmpData.StatusFlag.4 := WORD_TO_BOOL(MODBUS.MB_Resp.Data[4]);
				tmpData.StatusFlag.5 := WORD_TO_BOOL(MODBUS.MB_Resp.Data[5]);
				tmpData.StatusFlag.6 := WORD_TO_BOOL(MODBUS.MB_Resp.Data[6]);
				tmpData.StatusFlag.7 := WORD_TO_BOOL(MODBUS.MB_Resp.Data[7]);
				tmpData.StatusFlag.8 := WORD_TO_BOOL(MODBUS.MB_Resp.Data[8]);
				tmpData.StatusFlag.9 := WORD_TO_BOOL(MODBUS.MB_Resp.Data[9]);
				tmpData.StatusFlag.10 := WORD_TO_BOOL(MODBUS.MB_Resp.Data[10]);
				tmpData.StatusFlag.11 := WORD_TO_BOOL(MODBUS.MB_Resp.Data[11]);
				tmpData.StatusFlag.12 := WORD_TO_BOOL(MODBUS.MB_Resp.Data[12]);
				tmpData.StatusFlag.13 := WORD_TO_BOOL(MODBUS.MB_Resp.Data[13]);

				(* rinfresco il Watchdog dell' HVAC *)

				MODBUS.MB_Query.FunctionCode 		:= 16#10;
				MODBUS.MB_Query.Write_StartAddress	:= 1;
				MODBUS.MB_Query.Write_Quantity		:= 1;
				MODBUS.MB_Query.Write_Data[0] 		:= 5000;    	(* Questo valore deve essere costantemente rinfrescato in quanto
																		se va a zero l'HVAC va in allarme mancanza comunicazione
																		modBus mandando in stop *)

				MODBUS.MB_Start := TRUE;
				sta := 11;

			END_IF
		END_IF


	11:	(* Temperatura da Controllare : Temperatura ambiente	*)
		IF NOT MODBUS.MB_Start THEN
			IF MODBUS.MB_MASTER.MB_Error<>MB_NO_ERROR OR MODBUS.MB_Resp.Error<>0 THEN
				sta:=100;
			ELSE
				MODBUS.MB_Query.FunctionCode 		:= 16#10;
				MODBUS.MB_Query.Write_StartAddress	:= 20;
				MODBUS.MB_Query.Write_Quantity		:= 1;
				MODBUS.MB_Query.Write_Data[0]		:= INT_TO_WORD(SetBmsTenv); (* INT_TO_WORD(Data.Treturn); *)

				sta := 12;
			END_IF

    			MODBUS.MB_Start := TRUE;

		END_IF

	12:	(* Scrittura di temperatura del Set Point della macchina *)
		IF NOT MODBUS.MB_Start THEN
			IF MODBUS.MB_MASTER.MB_Error<>MB_NO_ERROR OR MODBUS.MB_Resp.Error<>0 THEN
				sta:=100;
			ELSE

				MODBUS.MB_Query.FunctionCode		:= 16#10;
				MODBUS.MB_Query.Write_StartAddress	:= 34;
				MODBUS.MB_Query.Write_Quantity		:= 16#1;
				MODBUS.MB_Query.Write_Data[0]		:= SetPointTemp;

				MODBUS.MB_Start := TRUE;
				sta := 13;
			END_IF
		END_IF

	13:	(* Write HVAC On/Off *)
		IF NOT MODBUS.MB_Start THEN
			IF MODBUS.MB_MASTER.MB_Error<>MB_NO_ERROR OR MODBUS.MB_Resp.Error<>0 THEN
				sta:=100;
			ELSE

				MODBUS.MB_Query.FunctionCode		:= 16#10;
				MODBUS.MB_Query.Write_StartAddress	:= 84;
				MODBUS.MB_Query.Write_Quantity		:= 16#1;
				MODBUS.MB_Query.Write_Data[0]		:= BOOL_TO_WORD(OnOff);

				MODBUS.MB_Start := TRUE;
				sta := 14;
			END_IF
		END_IF


	14:	(* Scrittura delle soglie per il controllo del CO2 - ppm Min e MAX*)
		IF fWriteLimitippmCO2 THEN
		IF NOT MODBUS.MB_Start THEN
			IF MODBUS.MB_MASTER.MB_Error<>MB_NO_ERROR OR MODBUS.MB_Resp.Error<>0 THEN
				sta:=100;
			ELSE

				MODBUS.MB_Query.FunctionCode		:= 16#10;
				MODBUS.MB_Query.Write_StartAddress	:= 187;
				MODBUS.MB_Query.Write_Quantity		:= 2;
				SogliaMinppmCO2:=LIMIT(SogliaMinppmCO2,0,LIMIT(SogliaMaxppmCO2,0,2000));
				MODBUS.MB_Query.Write_Data[0]		:= SogliaMinppmCO2 ; (* MinThrECO; *)
 				SogliaMaxppmCO2:=LIMIT(SogliaMaxppmCO2,MODBUS.MB_Query.Write_Data[0],2000);
				MODBUS.MB_Query.Write_Data[1]		:= SogliaMaxppmCO2; (* MaxThrECO;*)

				MODBUS.MB_Start := TRUE;
				fWriteLimitippmCO2:=FALSE;
				sta := 15;
			END_IF
		END_IF
		ELSE
				sta := 15;
		END_IF
	15: (* Scrittura delle soglie per il controllo del CO2 - Limite serranda min *)
		IF fWriteLimitiSerr THEN
		IF NOT MODBUS.MB_Start THEN
			IF MODBUS.MB_MASTER.MB_Error<>MB_NO_ERROR OR MODBUS.MB_Resp.Error<>0 THEN
				sta:=100;
			ELSE

				MODBUS.MB_Query.FunctionCode		:= 16#10;
				MODBUS.MB_Query.Write_StartAddress	:= 4;
				MODBUS.MB_Query.Write_Quantity		:= 1;
				SogliaMinimaSerrandaAria:=LIMIT(SogliaMinimaSerrandaAria,200,1000);
				MODBUS.MB_Query.Write_Data[0]		:=  SogliaMinimaSerrandaAria;

				MODBUS.MB_Start := TRUE;
				fWriteLimitiSerr:=FALSE;
				sta := 16;
			END_IF
		END_IF
		ELSE
				sta := 16;
		END_IF


	16: (* Scrittura Limiti per attivazione Free Cooling - Min e MAX *)
		IF fWriteAttivazioneFreeCooling THEN

		IF NOT MODBUS.MB_Start THEN
			IF MODBUS.MB_MASTER.MB_Error<>MB_NO_ERROR OR MODBUS.MB_Resp.Error<>0 THEN
				sta:=100;
			ELSE

				MODBUS.MB_Query.FunctionCode		:= 16#10;
				MODBUS.MB_Query.Write_StartAddress	:= 162;
				MODBUS.MB_Query.Write_Quantity		:= 2;
				MODBUS.MB_Query.Write_Data[0]		:= Intero_WORD(TempMinAttFreeCooling);
				MODBUS.MB_Query.Write_Data[1]		:= Intero_WORD(TempMaxAttFreeCooling);
				MODBUS.MB_Start := TRUE;
				fWriteAttivazioneFreeCooling:=FALSE;
				sta := 17;
			END_IF
		END_IF
		ELSE
				sta := 17;
		END_IF


	17:  (* Leggo lo stato della macchina *)

		IF NOT  MODBUS.MB_Start THEN
			MODBUS.MB_Query.SlaveAddress		:= ADDRESS;
			MODBUS.MB_Query.FunctionCode		:= 16#03;
			MODBUS.MB_Query.Read_StartAddress	:= 154;
			MODBUS.MB_Query.Read_Quantity		:= 3;

			MODBUS.MB_Start := TRUE;
			sta := 18;
		END_IF

	18:	IF NOT MODBUS.MB_Start THEN
			IF MODBUS.MB_MASTER.MB_Error<>MB_NO_ERROR OR MODBUS.MB_Resp.Error<>0 THEN
				sta:=100;
			ELSE
				MacchinaInRaffreddamento :=  MODBUS.MB_Resp.Data[0];
				MacchinaInZonaMorta :=  MODBUS.MB_Resp.Data[1];
				MacchinaInRiscaldamento :=  MODBUS.MB_Resp.Data[2];

				MODBUS.MB_Query.SlaveAddress		:= ADDRESS;
				MODBUS.MB_Query.FunctionCode		:= 16#03;
				MODBUS.MB_Query.Read_StartAddress	:= 2;
				MODBUS.MB_Query.Read_Quantity		:= 4;

				MODBUS.MB_Start := TRUE;

				sta := 19;
			END_IF
		END_IF


	19:
		IF NOT MODBUS.MB_Start THEN
			IF MODBUS.MB_MASTER.MB_Error<>MB_NO_ERROR OR MODBUS.MB_Resp.Error<>0 THEN
				sta:=100;
			ELSE


					ReadSetPointColdDay :=  MODBUS.MB_Resp.Data[0];
					ReadSetPointHeatDay :=  MODBUS.MB_Resp.Data[1];
					ReadSogliaMinimaSerrandaAria :=  MODBUS.MB_Resp.Data[2];

					MODBUS.MB_Query.SlaveAddress		:= ADDRESS;
					MODBUS.MB_Query.FunctionCode		:= 16#03;
					MODBUS.MB_Query.Read_StartAddress	:= 187;
					MODBUS.MB_Query.Read_Quantity		:= 2;

					MODBUS.MB_Start := TRUE;

				sta := 20;
			END_IF
		END_IF

	20: (* Leggo le soglie di ppm impostata nella macchiana*)
		IF NOT MODBUS.MB_Start THEN
			IF MODBUS.MB_MASTER.MB_Error<>MB_NO_ERROR OR MODBUS.MB_Resp.Error<>0 THEN
				sta:=100;
			ELSE


					ReadSogliaMinppmCO2 :=  MODBUS.MB_Resp.Data[0];
					ReadSogliaMaxppmCO2 :=  MODBUS.MB_Resp.Data[1];

					MODBUS.MB_Query.SlaveAddress		:= ADDRESS;
					MODBUS.MB_Query.FunctionCode		:= 16#03;
					MODBUS.MB_Query.Read_StartAddress	:= 91;
					MODBUS.MB_Query.Read_Quantity		:= 1;

					MODBUS.MB_Start := TRUE;

				sta := 21;
			END_IF
		END_IF

	21:	(* Scrivo il valre set 	Set Point di Temperatura modalità riscaldamento in °C
								Set Point di Temperatura modalità raffreddamento in °C	*)
		IF NOT MODBUS.MB_Start THEN
			IF MODBUS.MB_MASTER.MB_Error<>MB_NO_ERROR OR MODBUS.MB_Resp.Error<>0 THEN
				sta:=100;
			ELSE

					MODBUS.MB_Query.FunctionCode 		:= 16#10;
					MODBUS.MB_Query.Write_StartAddress	:= 2;
					MODBUS.MB_Query.Write_Quantity		:= 2;
					MODBUS.MB_Query.Write_Data[0] 		:= LIMIT((SetPointTemp + SetPointColdDay),80,350);
					MODBUS.MB_Query.Write_Data[1] 		:= LIMIT((SetPointTemp - SetPointHeatDay),80,350);
					MODBUS.MB_Start := TRUE;

				sta :=22;
			END_IF
		END_IF


	22:	(* Lettura stato soglie impostate per la gestione del Free Cooling *)
		IF NOT MODBUS.MB_Start THEN
			IF MODBUS.MB_MASTER.MB_Error<>MB_NO_ERROR OR MODBUS.MB_Resp.Error<>0 THEN
				sta:=100;
			ELSE

				MODBUS.MB_Query.SlaveAddress		:= ADDRESS;
				MODBUS.MB_Query.FunctionCode		:= 16#03;
				MODBUS.MB_Query.Read_StartAddress	:= 162;
				MODBUS.MB_Query.Read_Quantity		:= 2;


				MODBUS.MB_Start := TRUE;
				sta := 23;
			END_IF
		END_IF

	23:	(* Lettura stato soglie impostate per la gestione del Free Cooling *)
		IF NOT MODBUS.MB_Start THEN
			IF MODBUS.MB_MASTER.MB_Error<>MB_NO_ERROR OR MODBUS.MB_Resp.Error<>0 THEN
				sta:=100;
			ELSE

					ReadTempMinAttFreeCooling := Word_Intero( MODBUS.MB_Resp.Data[0]);
					ReadTempMaxAttFreeCooling :=  MODBUS.MB_Resp.Data[1];

					MODBUS.MB_Query.SlaveAddress		:= ADDRESS;
					MODBUS.MB_Query.FunctionCode		:= 16#03;
					MODBUS.MB_Query.Read_StartAddress	:= 91;
					MODBUS.MB_Query.Read_Quantity		:= 1;

					MODBUS.MB_Start := TRUE;
				sta := 24;
			END_IF
		END_IF


	24:	(* Lettura stato Free Cooling attivato - Disattivato *)
		IF NOT MODBUS.MB_Start THEN
			IF MODBUS.MB_MASTER.MB_Error<>MB_NO_ERROR OR MODBUS.MB_Resp.Error<>0 THEN
				sta:=100;
			ELSE

					ReadStatoAttivaFreeCooling := MODBUS.MB_Resp.Data[0];

			(*
					MODBUS.MB_Query.SlaveAddress		:= ADDRESS;
					MODBUS.MB_Query.FunctionCode		:= 16#03;
					MODBUS.MB_Query.Read_StartAddress	:= 91;
					MODBUS.MB_Query.Read_Quantity		:= 1;
			
					MODBUS.MB_Start := TRUE; *)
				sta := 25;
			END_IF
		END_IF


	25: (* Scrittura Abuilitazioni Set Point Giorno e Notte *)
		IF fWriteAttivazioneSetPoint THEN

		IF NOT MODBUS.MB_Start THEN
			IF MODBUS.MB_MASTER.MB_Error<>MB_NO_ERROR OR MODBUS.MB_Resp.Error<>0 THEN
				sta:=100;
			ELSE


				MODBUS.MB_Query.FunctionCode		:= 16#10;
				MODBUS.MB_Query.Write_StartAddress	:= 86;
				MODBUS.MB_Query.Write_Quantity		:= 4;
				MODBUS.MB_Query.Write_Data[0]		:= WriteBMSGiornoAttivazione;
				MODBUS.MB_Query.Write_Data[1]		:= WriteBMSGiornoAttivazioneZM;
				MODBUS.MB_Query.Write_Data[2]		:= WriteBMSNotteAttivazione;
				MODBUS.MB_Query.Write_Data[3]		:= WriteBMSNotteAttivazioneZM;

				MODBUS.MB_Start := TRUE;
				fWriteAttivazioneSetPoint:=FALSE;
				sta := 26;
			END_IF
		END_IF
		ELSE
				sta := 26;
		END_IF

	26:	(* Lettura stato soglie impostate per la gestione del Free Cooling *)
		IF NOT MODBUS.MB_Start THEN
			IF MODBUS.MB_MASTER.MB_Error<>MB_NO_ERROR OR MODBUS.MB_Resp.Error<>0 THEN
				sta:=100;
			ELSE
					MODBUS.MB_Query.SlaveAddress		:= ADDRESS;
					MODBUS.MB_Query.FunctionCode		:= 16#03;
					MODBUS.MB_Query.Read_StartAddress	:= 86;
					MODBUS.MB_Query.Read_Quantity		:= 4;

					MODBUS.MB_Start := TRUE;
				sta := 27;
			END_IF
		END_IF


	27:	(* Lettura stato Free Cooling attivato - Disattivato *)
		IF NOT MODBUS.MB_Start THEN
			IF MODBUS.MB_MASTER.MB_Error<>MB_NO_ERROR OR MODBUS.MB_Resp.Error<>0 THEN
				sta:=100;
			ELSE

					ReadBMSGiornoAttivazione := MODBUS.MB_Resp.Data[0];
					ReadBMSGiornoAttivazioneZM := MODBUS.MB_Resp.Data[1];
					ReadBMSNotteAttivazione := MODBUS.MB_Resp.Data[2];
					ReadBMSNotteAttivazioneZM := MODBUS.MB_Resp.Data[3];

			(*
					MODBUS.MB_Query.SlaveAddress		:= ADDRESS;
					MODBUS.MB_Query.FunctionCode		:= 16#03;
					MODBUS.MB_Query.Read_StartAddress	:= 91;
					MODBUS.MB_Query.Read_Quantity		:= 1;
			
					MODBUS.MB_Start := TRUE; *)
				sta := 50;
			END_IF
		END_IF




	50:	IF NOT MODBUS.MB_Start THEN
			IF MODBUS.MB_MASTER.MB_Error<>MB_NO_ERROR OR MODBUS.MB_Resp.Error<>0 THEN
				sta:=100;
			ELSE
				(* Copy temporary read data *)
				MEMCPY(ADR(tmpData), ADR(Data), SIZEOF(Data));


				fModbusAlr := FALSE;
				MODBUS.MB_Lock := FALSE;
				sta := 0;
			END_IF
		END_IF











	100: (* === Check MODBUS error *)
		(* Release MODBUS *)
		MODBUS.MB_Lock := FALSE;

		(* Retries *)
		retry := retry+1;

		IF retry>3 THEN
			retry := 0;

			(* Signal event *)
			IF Status_Log<>2 THEN
				LogEv(EL_Alarm,EO_HVAC,ID,2,SEL(ModBus.MB_MASTER.MB_Error<>0,'0','1'));
			END_IF
			fModbusAlr := TRUE;
		END_IF

		sta := 0;

ELSE
	sta := 0;
END_CASE
END_ACTION

(* POU Plant_Objects/obj_MODBUS, ST *)
FUNCTION_BLOCK obj_MODBUS
(* === MODBUS PROTOCOL INTERFACE ===
   v1.1[19/06/15] - Added new VARS allocation and searching
*)
VAR CONSTANT
	VARS_Max	: BYTE := 32;
END_VAR
VAR_INPUT
	(* Settings *)
	ID			: BYTE;
	COM			: BYTE;
	BAUDRATE	: COM_BAUDRATE;
	RS485		: BOOL := FALSE;

	(* Interface *)
	MB_MASTER	: MODBUS_EXTENDED_MASTER;
	MB_Start	: BOOL;
	MB_Query	: typModbusExtendedQuery;
	MB_Resp		: typModbusResponse;
	MB_Lock		: BOOL;

	(* Variables management *)
	VARS_En		: BOOL;
	VARS		: ARRAY [0..VARS_Max] OF typ_MODBUS_VAR;
	VARS_Check	: BOOL;
	VARS_Alarm	: BOOL;

	(* Variables allocation *)
	VAR_Pointer : POINTER TO ARRAY[0..99] OF WORD;
	VAR_Cfg		: POINTER TO typ_MODBUS_VAR;
END_VAR
VAR_OUTPUT
	(* Status *)
	Status_Log	: BYTE;
	Status_Vis	: DWORD;
END_VAR
VAR
	sta         : BYTE :=0;
	i			: BYTE;
	j			: BYTE;
	Alarm		: FLT_EVENT := (INITEV:=FALSE);

	VarTmr		: TON := (PT:=T#1s);
	VarSta		: BYTE; (* Status *)
	VarCnt		: BYTE; (* Scan counter *)
	VarRetry	: BYTE;
	VarAlarm	: BYTE; (* Last variable with errors *)
END_VAR
(* NB: Timeout has been changed: 750ms instead of 250ms as usual. This because Frer declares
       "Minimum response time-out (to be set on the master): 500ms." 		*)
MB_MASTER(ENABLE:=TRUE,	ASCII_Mode:=FALSE, bCOM_PORT:=COM, cbCOM_BAUDRATE:=BAUDRATE, cpCOM_PARITY:=PARITY_NO,
		csCOM_STOPBITS:=STOPBITS_2,	cbsCOM_BYTESIZE:=BS_8, cfCOM_FLOW_CONTROL:=SEL(RS485,NO_FLOW_CONTROL,HALFDUPLEX),
		tTIME_OUT:=t#250ms,	StartFunction:=MB_Start, ExtQuery:=MB_Query, Response:=MB_Resp);

(* Process variable management *)
IF VARS_En THEN VARS_Process(); END_IF

(* Check status *)
Alarm(IN:=(MB_MASTER.bInterfaceError<>0));
IF Alarm.EVH THEN
	LogEv(SEL(MB_MASTER.bInterfaceError<>3,EL_Wrn,EL_Alarm),EO_MODBUS,ID,1,BYTE_TO_STRING(MB_MASTER.bInterfaceError));
END_IF
IF Alarm.EVL THEN								(* Trigger a fall edge: MODBUS back working *)
	LogEv(EL_Log,EO_MODBUS,ID,2,'MODBUS_OK');
END_IF

(* Log/visu status *)
   IF Alarm.IN   THEN Status_Log:=2; Status_Vis:=COLOR_RED;
ELSIF Vars_Alarm THEN Status_Log:=1; Status_Vis:=COLOR_YELLOW;
  				 ELSE Status_Log:=0; Status_Vis:=COLOR_GREEN;
END_IF
END_FUNCTION_BLOCK
ACTION VAR_Search:
(* Search VAR with specific pointer if not found return first free VAR
	[Last VAR is not active... used as safe area...] 
*)
j:=VARS_Max;
FOR i := 0 TO VARS_Max-1 DO
	IF VARS[i].Variable=0 AND j>i THEN j:=i; END_IF
	IF VARS[i].Variable=VAR_Pointer THEN
		VAR_Cfg:=ADR(VARS[i]);
		RETURN;
	END_IF
END_FOR
VAR_Cfg:=ADR(VARS[j]);
END_ACTION
ACTION VARS_Process:
(* Update var timers *)
VarTmr(IN:=(NOT VarTmr.Q));
IF VarTmr.Q THEN
	FOR i := 0 TO VARS_Max DO
		IF VARS[i].Refresh_Cnt>0 THEN VARS[i].Refresh_Cnt:=VARS[i].Refresh_Cnt-1; END_IF
	END_FOR
	VARS_Check:=TRUE;
END_IF


(* Process status *)
CASE VarSta OF
	0: (* === Init *)
		VarCnt:=0;
		VarSta:=1;

	1: (* === Wait check signal *)
		IF VARS_Check THEN				(* Decremented "Refresh_Cnt" *)
			VARS_Check:=FALSE;
			VarCnt:=0;
			VarSta:=2;
		END_IF

	2: (* === Check loop *)
		IF NOT (MB_Lock OR MB_Start) THEN
			WHILE VarCnt<=(VARS_Max-1) AND VarSta=2 DO
				(* Check only active vars *)
				IF VARS[VarCnt].Variable<>0 THEN			(* "Variable" is a pointer to word, so if 0 no address *)
					(* Check var auto-refresh on timer checks *)
					IF VARS[VarCnt].Refresh_Time>0 AND VARS[VarCnt].Refresh_Cnt=0 THEN
						VARS[VarCnt].Refresh_Cnt:=VARS[VarCnt].Refresh_Time;
						VarSta:=3;
					END_IF
					(* Check refresh for change or request *)
					CASE VARS[VarCnt].FunCode OF
						5,6,15,16: (* Write functions *)
							IF VARS[VarCnt].Variable_Size=1 THEN
								IF VARS[VarCnt].Variable^<>VARS[VarCnt].Variable_Mirror THEN
									VARS[VarCnt].Variable_Mirror:=VARS[VarCnt].Variable^;
									VarSta:=3;
								END_IF
							ELSE
								IF VARS[VarCnt].Variable_Mirror<>0 THEN
									VARS[VarCnt].Variable_Mirror:=0;
									VarSta:=3;
								END_IF
							END_IF
						1,2,3,4: (* Read functions *)
							IF VARS[VarCnt].Variable_Mirror<>0 THEN
								VARS[VarCnt].Variable_Mirror:=0;
								VarSta:=3;
							END_IF
					END_CASE
				END_IF
				(* Process query *)
				IF VarSta=3 THEN
					MB_Lock:=TRUE;
					MB_Query.SlaveAddress:=VARS[VarCnt].SlaveAddress;
					MB_Query.FunctionCode:=VARS[VarCnt].FunCode;
					CASE VARS[VarCnt].FunCode OF
						16#5,16#6,16#F,16#10:
							MB_Query.Read_Quantity:=0;
							MB_Query.Read_StartAddress:=0;
							MB_Query.Write_StartAddress:=VARS[VarCnt].FunAddress;
							MB_Query.Write_Quantity:=VARS[VarCnt].Variable_Size;
							IF VARS[VarCnt].Variable_Size=200 THEN
								COPY_32SWAP16(VARS[VarCnt].Variable, ADR(MB_Query.Write_Data[0]));
							ELSIF VARS[VarCnt].Variable_Size>1 THEN
								MEMCPY(VARS[VarCnt].Variable, ADR(MB_Query.Write_Data[0]), 2*VARS[VarCnt].Variable_Size);
							ELSE
								MB_Query.Write_Data[0]:=VARS[VarCnt].Variable^;
							END_IF
						16#1,16#2,16#3,16#4:
							MB_Query.Read_StartAddress:=VARS[VarCnt].FunAddress;
							IF VARS[VarCnt].Variable_Size=200 THEN MB_Query.Read_Quantity:=2; ELSE		(* 200 -->> DWORD 32bits *)
							  MB_Query.Read_Quantity:=VARS[VarCnt].Variable_Size;
							END_IF
							MB_Query.Write_StartAddress:=0;
							MB_Query.Write_Quantity:=0;
					END_CASE
					VarRetry:=0;
					MB_Start:=TRUE;
				ELSE
					VarCnt:=VarCnt+1;
				END_IF
			END_WHILE
			(* Check loop completed -> no actions *)
			IF VarSta=2 THEN VarSta:=1; END_IF
		END_IF

	3: (* === Wait & process MB response *)
		IF NOT MB_Start THEN
			IF MB_MASTER.MB_Error=0 THEN
				CASE VARS[VarCnt].FunCode OF
					1,2,3,4:
						IF VARS[VarCnt].Variable_Size=200 THEN
							COPY_32SWAP16(ADR(MB_Resp.Data), VARS[VarCnt].Variable);
						ELSIF VARS[VarCnt].Variable_Size>1 THEN
							MEMCPY(ADR(MB_Resp.Data), VARS[VarCnt].Variable, 2*VARS[VarCnt].Variable_Size);
						ELSE
							VARS[VarCnt].Variable^:=MB_Resp.Data[0];
						END_IF
				END_CASE
				MB_Lock:=FALSE;
				(* Signal error recovery *)
				IF VARS_Alarm=TRUE AND VarCnt=VarAlarm THEN
					LogEv(EL_Wrn,EO_MODBUS,ID,5,'');
					VARS_Alarm:=FALSE;
				END_IF
				(* Next var *)
				VarCnt:=VarCnt+1;
				VarSta:=2;
			ELSE
				IF VarRetry<3 THEN
					VarRetry:=VarRetry+1;
					MB_Start:=TRUE;
				ELSE
					MB_Lock:=FALSE;
					(* Signal error *)
					IF VARS_Alarm=FALSE THEN
						LogEv(EL_Wrn,EO_MODBUS,ID,3,INT_TO_STRING(MB_MASTER.MB_Error));
						VARS_Alarm:=TRUE;
						VarAlarm:=VarCnt-1;
					END_IF
					(* Next var *)
					VarCnt:=VarCnt+1;
					VarSta:=2;
				END_IF
			END_IF
		END_IF

ELSE
	VarSta:=0;
END_CASE
END_ACTION

(* POU Utils Functions/Word_Intero, ST *)
FUNCTION Word_Intero : INT
VAR_INPUT
	IN_WORD: WORD;
END_VAR
VAR
	Appoggio:DWORD;
END_VAR
IF IN_WORD>32766 THEN
	Appoggio:= (65534 - IN_WORD);
	Word_Intero:= -(DWORD_TO_INT(Appoggio));
ELSE
	Word_Intero:= WORD_TO_INT(IN_WORD);
END_IF
END_FUNCTION

(* POU Plant_Objects/obj_LUXM, ST *)
FUNCTION_BLOCK obj_LUXM
(* === Metered ON/OFF Illumination Point ===
   Failure detection:
   Statistic data:
   
   - Come identifico l'assenza del nodo?? (Rele non funzionante/non alimentato)
   - Acquisizione carico dopo accensione?? Dati carico in NVM!
   
   v1.0[07/05/15] - Create
*)
VAR_INPUT
	(* Settings *)
	ID				: BYTE;
	(* Controls *)
	CTRL_MODE		: INT;  (* 0:MAN OFF, -1:MAN-ON,
							   -2:KEY-ON, -3:KEY-OFF, -4:DAY, -5:NIGHT,
							   N>0:Nsec-TIMER *)
	CTRL_TRIG		: BOOL; (* Trigger for timer start *)
	CTRL_KEY		: BOOL; (* External KEY control input *)
	CTRL_SENS		: BOOL; (* External dark sensor input [1:Dark] *)
	CTRL_EXTON		: BOOL; (* External forced activation *)
	(* Physical inputs *)
	REL_ST			: BOOL; (* Status feedback *)
	REL_V			: WORD; (* [E-1 V] Voltage *)
	REL_A			: WORD; (* [E-1 A] Current *)
	REL_ALM			: WORD; (* Error status [0:OK, 1:Disconnected, 2:LoadLOW, 3:LoadHIGH, 4:Overload, 5:ControlFAIL] *)
	REL_TEMP		: INT;  (* [E-1 °C] Temperature *)
	REL_TON			: DWORD;(* [sec] External working time counter *)  
	(* Persistent *)(*
	WORKINGTIME		: POINTER TO DWORD; (* [sec] Internal working time counter *)
	POWERONCYCLES	: POINTER TO DWORD; (* Internal counter of power-on cycles *)
	ENERGYCOUNTER	: POINTER TO DWORD; (* [E-1 kWh] Internal energy counter *)
	ENERGYCOUNTER_T : POINTER TO DWORD; (* Temporary energy in E-2*Wsec *)*)
END_VAR
VAR_IN_OUT
	WORKINGTIME		: DWORD; (* [sec] Internal working time counter *)
	POWERONCYCLES	: DWORD; (* Internal counter of power-on cycles *)
	ENERGYCOUNTER	: DWORD; (* [E-1 kWh] Internal energy counter *)
	ENERGYCOUNTER_T : DWORD; (* Temporary energy in E-2*Wsec *)
END_VAR
VAR_OUTPUT
	(* Physical outputs *)
	REL_EN			: BOOL;	(* Control output *)
	(* Status *)
	Status_Log		: BYTE;
	Status_Vis 		: DWORD;
END_VAR
VAR
	TickTimer		: TON := ( PT:=T#1S );
	TrigTimer		: TOF;
	sREL_EN			: FLT_EVENT;
	sREL_ALM		: WORD:=16#FFFF;
	chkREL_ST		: FLT_TIME := ( TTAP:=T#20S, INITEV:=FALSE );
END_VAR
(* Trig timer *)
TrigTimer(IN:=CTRL_TRIG);

(* Control logic *)
IF CTRL_EXTON THEN
	REL_EN:=TRUE;
ELSE
	CASE CTRL_MODE OF
		 0: REL_EN:=FALSE;
		-1: REL_EN:=TRUE;
		-2: REL_EN:=CTRL_KEY;
		-3: REL_EN:=NOT CTRL_KEY;
		-4: REL_EN:=CTRL_SENS;
		-5: REL_EN:=NOT CTRL_SENS;
	ELSE
		IF CTRL_MODE>0 THEN
			REL_EN:=TrigTimer.Q;
			TrigTimer.PT:=T#1S*CTRL_MODE;
		ELSE
			REL_EN:=FALSE;
		END_IF
	END_CASE
END_IF

(* Temporary energy counter *)
TickTimer(IN:=NOT TickTimer.Q);
IF TickTimer.Q AND REL_EN THEN
	WORKINGTIME:=WORKINGTIME+1;
	ENERGYCOUNTER_T:=ENERGYCOUNTER_T+REL_V*REL_A;
	IF ENERGYCOUNTER_T>36000000 THEN
		ENERGYCOUNTER_T:=ENERGYCOUNTER_T-36000000;
		ENERGYCOUNTER:=ENERGYCOUNTER+1;		
	END_IF
END_IF

(* Generate status events *)
sREL_EN(IN:=REL_EN);
IF sREL_EN.EVL THEN LogEv(EL_Log,EO_LUXM,ID,2,''); END_IF
IF sREL_EN.EVH THEN LogEv(EL_Log,EO_LUXM,ID,3,''); POWERONCYCLES:=POWERONCYCLES+1; END_IF

(* Check status feedback *)
chkREL_ST(IN:=(REL_ST<>REL_EN));
IF chkREL_ST.EVH THEN LogEv(EL_Alarm,EO_LUXM,ID,9,''); END_IF
IF chkREL_ST.EVL AND sREL_ALM=0 THEN LogEv(EL_Log,EO_LUXM,ID,1,''); END_IF

(* Check controller alarm *)
IF sREL_ALM<>REL_ALM THEN
	CASE REL_ALM OF
		0: IF NOT chkREL_ST.OUT THEN LogEv(EL_Log,EO_LUXM,ID,1,''); END_IF
		1: LogEv(EL_Alarm,EO_LUXM,ID,6,'');
		2: LogEv(EL_Wrn  ,EO_LUXM,ID,4,WORD_TO_STRING(REL_A));
		3: LogEv(EL_Wrn  ,EO_LUXM,ID,5,WORD_TO_STRING(REL_A));
		4: LogEv(EL_Alarm,EO_LUXM,ID,7,WORD_TO_STRING(REL_A));
		5: LogEv(EL_Alarm,EO_LUXM,ID,8,'');
	END_CASE
	sREL_ALM:=REL_ALM;
END_IF

(* Status color *)
   IF REL_ALM=1 OR REL_ALM>3 OR chkREL_ST.OUT	THEN Status_Log:=2; Status_Vis:=COLOR_RED;
ELSIF REL_ALM<>0								THEN Status_Log:=1; Status_Vis:=COLOR_YELLOW;
                  	   							ELSE Status_Log:=0; Status_Vis:=SEL(REL_EN,COLOR_GREEN_OFF,COLOR_GREEN);
END_IF
END_FUNCTION_BLOCK
ACTION AddLogData:
Logger.s1:=INSERT('&LUXM=',BYTE_TO_STRING(ID),5);
IF ID<10 THEN Logger.s1:=INSERT(Logger.s1,'0',5); END_IF

Logger.s1:=CONCAT(Logger.s1,WORD_TO_STRING(REL_V));				Logger.s1:=CONCAT(Logger.s1,';');
Logger.s1:=CONCAT(Logger.s1,WORD_TO_STRING(REL_A));				Logger.s1:=CONCAT(Logger.s1,';');
Logger.s1:=CONCAT(Logger.s1,DWORD_TO_STRING(ENERGYCOUNTER));	Logger.s1:=CONCAT(Logger.s1,';');
Logger.s1:=CONCAT(Logger.s1,DWORD_TO_STRING(WORKINGTIME));		Logger.s1:=CONCAT(Logger.s1,';');
Logger.s1:=CONCAT(Logger.s1,DWORD_TO_STRING(POWERONCYCLES));	Logger.s1:=CONCAT(Logger.s1,';');
Logger.s1:=CONCAT(Logger.s1,INT_TO_STRING(REL_TEMP));			Logger.s1:=CONCAT(Logger.s1,';');

Logger.s1:=CONCAT(Logger.s1,BYTE_TO_STRING(Status_Log));
ADDSTRING(ADR(Logger.TData), ADR(Logger.s1), Logger.TLen);
END_ACTION
ACTION StatReset:
(* Reset statistic counters *)
WORKINGTIME:=0;
POWERONCYCLES:=0;
ENERGYCOUNTER:=0;
END_ACTION

(* POU Plant_Objects/obj_LUXP, ST *)
FUNCTION_BLOCK obj_LUXP
(* === Metered ON/OFF Illumination Point ===
   Failure detection:
   Statistic data:
   
